    |   movel([0.686921, -1.277827, -2.632564, -0.801997, 1.570796, 2.257718],accel_mss,speed_ms,0,blend_radius_m)
    |   speed_ms = 0.040
    |   movel([0.686153, -1.291546, -2.624638, -0.796205, 1.570796, 2.256949],accel_mss,speed_ms,0,blend_radius_m)
    |   speed_ms = 0.005
    |   movel([0.686153, -1.300886, -2.628985, -0.782518, 1.570796, 2.256949],accel_mss,speed_ms,0,blend_radius_m)
    |   speed_ms = 0.025
    |   movel([0.686563, -1.298464, -2.630421, -0.783504, 1.570796, 2.257359],accel_mss,speed_ms,0,blend_radius_m)
    |   movel([0.686602, -1.296181, -2.631767, -0.784440, 1.570796, 2.257399],accel_mss,speed_ms,0,blend_radius_m)
    |   movel([0.686283, -1.294070, -2.633007, -0.785312, 1.570796, 2.257079],accel_mss,speed_ms,0,blend_radius_m)
    |   movel([0.685611, -1.292156, -2.634126, -0.786108, 1.570796, 2.256407],accel_mss,speed_ms,0,blend_radius_m)
    |   movel([0.684603, -1.290473, -2.635106, -0.786811, 1.570796, 2.255399],accel_mss,speed_ms,0,blend_radius_m)
    |   movel([0.683264, -1.289050, -2.635931, -0.787408, 1.570796, 2.254061],accel_mss,speed_ms,0,blend_radius_m)
    |   movel([0.681611, -1.287921, -2.636584, -0.787884, 1.570796, 2.252407],accel_mss,speed_ms,0,blend_radius_m)
    |   movel([0.679652, -1.287111, -2.637052, -0.788226, 1.570796, 2.250448],accel_mss,speed_ms,0,blend_radius_m)
    |   movel([0.677407, -1.286654, -2.637315, -0.788420, 1.570796, 2.248203],accel_mss,speed_ms,0,blend_radius_m)
    |   movel([0.674916, -1.286573, -2.637362, -0.788454, 1.570796, 2.245712],accel_mss,speed_ms,0,blend_radius_m)
    |   movel([0.672268, -1.286884, -2.637182, -0.788322, 1.570796, 2.243064],accel_mss,speed_ms,0,blend_radius_m)
    |   movel([0.669552, -1.287613, -2.636762, -0.788014, 1.570796, 2.240348],accel_mss,speed_ms,0,blend_radius_m)
    |   movel([0.666852, -1.288777, -2.636089, -0.787523, 1.570796, 2.237648],accel_mss,speed_ms,0,blend_radius_m)
    |   movel([0.665538, -1.289527, -2.635654, -0.787208, 1.570796, 2.236335],accel_mss,speed_ms,0,blend_radius_m)
    |   movel([0.664263, -1.290390, -2.635154, -0.786846, 1.570796, 2.235059],accel_mss,speed_ms,0,blend_radius_m)
    |   movel([0.663035, -1.291369, -2.634584, -0.786436, 1.570796, 2.233831],accel_mss,speed_ms,0,blend_radius_m)
    |   movel([0.661866, -1.292469, -2.633943, -0.785977, 1.570796, 2.232663],accel_mss,speed_ms,0,blend_radius_m)
    |   movel([0.660768, -1.293687, -2.633231, -0.785471, 1.570796, 2.231564],accel_mss,speed_ms,0,blend_radius_m)
    |   movel([0.659756, -1.295024, -2.632448, -0.784917, 1.570796, 2.230552],accel_mss,speed_ms,0,blend_radius_m)
    |   speed_ms = 0.005
    |   movel([0.659756, -1.285649, -2.628074, -0.798666, 1.570796, 2.230552],accel_mss,speed_ms,0,blend_radius_m)
    |   speed_ms = 0.040
    |   movel([0.667434, -1.296086, -2.621962, -0.794341, 1.570796, 2.238230],accel_mss,speed_ms,0,blend_radius_m)
    |   speed_ms = 0.005
    |   movel([0.667434, -1.305400, -2.626288, -0.780701, 1.570796, 2.238230],accel_mss,speed_ms,0,blend_radius_m)
    |   speed_ms = 0.025
    |   movel([0.669418, -1.304874, -2.626604, -0.780911, 1.570796, 2.240215],accel_mss,speed_ms,0,blend_radius_m)
    |   movel([0.671310, -1.304654, -2.626736, -0.781000, 1.570796, 2.242106],accel_mss,speed_ms,0,blend_radius_m)
    |   movel([0.673092, -1.304715, -2.626699, -0.780975, 1.570796, 2.243888],accel_mss,speed_ms,0,blend_radius_m)
    |   movel([0.674741, -1.305035, -2.626507, -0.780847, 1.570796, 2.245537],accel_mss,speed_ms,0,blend_radius_m)
    |   movel([0.676240, -1.305588, -2.626175, -0.780626, 1.570796, 2.247036],accel_mss,speed_ms,0,blend_radius_m)
    |   movel([0.677570, -1.306343, -2.625722, -0.780325, 1.570796, 2.248366],accel_mss,speed_ms,0,blend_radius_m)
    |   movel([0.678716, -1.307277, -2.625159, -0.779953, 1.570796, 2.249512],accel_mss,speed_ms,0,blend_radius_m)
    |   movel([0.679657, -1.308360, -2.624505, -0.779524, 1.570796, 2.250453],accel_mss,speed_ms,0,blend_radius_m)
    |   movel([0.680469, -1.309890, -2.623579, -0.778920, 1.570796, 2.251265],accel_mss,speed_ms,0,blend_radius_m)
    |   movel([0.680812, -1.311531, -2.622583, -0.778276, 1.570796, 2.251609],accel_mss,speed_ms,0,blend_radius_m)
    |   movel([0.680741, -1.313269, -2.621523, -0.777597, 1.570796, 2.251537],accel_mss,speed_ms,0,blend_radius_m)
    |   movel([0.680298, -1.315090, -2.620408, -0.776890, 1.570796, 2.251095],accel_mss,speed_ms,0,blend_radius_m)
    |   movel([0.679538, -1.316977, -2.619249, -0.776163, 1.570796, 2.250334],accel_mss,speed_ms,0,blend_radius_m)
    |   movel([0.678505, -1.318918, -2.618051, -0.775419, 1.570796, 2.249301],accel_mss,speed_ms,0,blend_radius_m)
    |   movel([0.677248, -1.320898, -2.616825, -0.774666, 1.570796, 2.248044],accel_mss,speed_ms,0,blend_radius_m)
    |   movel([0.675817, -1.322904, -2.615576, -0.773908, 1.570796, 2.246614],accel_mss,speed_ms,0,blend_radius_m)
    |   speed_ms = 0.005
    |   movel([0.675817, -1.313698, -2.611330, -0.787361, 1.570796, 2.246614],accel_mss,speed_ms,0,blend_radius_m)
    |   speed_ms = 0.040
    |   movel([0.665940, -1.309142, -2.614119, -0.789128, 1.570796, 2.236737],accel_mss,speed_ms,0,blend_radius_m)
    |   speed_ms = 0.005
    |   movel([0.665940, -1.318376, -2.618386, -0.775626, 1.570796, 2.236737],accel_mss,speed_ms,0,blend_radius_m)
    |   speed_ms = 0.025
    |   movel([0.667189, -1.319166, -2.617898, -0.775325, 1.570796, 2.237985],accel_mss,speed_ms,0,blend_radius_m)
    |   movel([0.668210, -1.320110, -2.617314, -0.774965, 1.570796, 2.239007],accel_mss,speed_ms,0,blend_radius_m)
    |   movel([0.669011, -1.321200, -2.616637, -0.774552, 1.570796, 2.239807],accel_mss,speed_ms,0,blend_radius_m)
    |   movel([0.669605, -1.322415, -2.615881, -0.774093, 1.570796, 2.240401],accel_mss,speed_ms,0,blend_radius_m)
    |   movel([0.670000, -1.323744, -2.615052, -0.773593, 1.570796, 2.240796],accel_mss,speed_ms,0,blend_radius_m)
    |   movel([0.670206, -1.325167, -2.614162, -0.773060, 1.570796, 2.241002],accel_mss,speed_ms,0,blend_radius_m)
    |   movel([0.670235, -1.326674, -2.613216, -0.772499, 1.570796, 2.241031],accel_mss,speed_ms,0,blend_radius_m)
    |   movel([0.670092, -1.328248, -2.612225, -0.771916, 1.570796, 2.240888],accel_mss,speed_ms,0,blend_radius_m)
    |   movel([0.669791, -1.329876, -2.611196, -0.771317, 1.570796, 2.240588],accel_mss,speed_ms,0,blend_radius_m)
    |   movel([0.669343, -1.331542, -2.610139, -0.770707, 1.570796, 2.240139],accel_mss,speed_ms,0,blend_radius_m)
    |   movel([0.668753, -1.333234, -2.609063, -0.770092, 1.570796, 2.239550],accel_mss,speed_ms,0,blend_radius_m)
    |   movel([0.668036, -1.334937, -2.607975, -0.769477, 1.570796, 2.238832],accel_mss,speed_ms,0,blend_radius_m)
    |   movel([0.667196, -1.336639, -2.606884, -0.768866, 1.570796, 2.237993],accel_mss,speed_ms,0,blend_radius_m)
    |   movel([0.665195, -1.339980, -2.604731, -0.767678, 1.570796, 2.235992],accel_mss,speed_ms,0,blend_radius_m)
    |   movel([0.664049, -1.341596, -2.603683, -0.767109, 1.570796, 2.234845],accel_mss,speed_ms,0,blend_radius_m)
    |   movel([0.664256, -1.341009, -2.604065, -0.767316, 1.570796, 2.235052],accel_mss,speed_ms,0,blend_radius_m)
    |   speed_ms = 0.005
    |   movel([0.664256, -1.331920, -2.599899, -0.780569, 1.570796, 2.235052],accel_mss,speed_ms,0,blend_radius_m)
    |   speed_ms = 0.040
    |   movel([0.669329, -1.341680, -2.593594, -0.777115, 1.570796, 2.240125],accel_mss,speed_ms,0,blend_radius_m)
    |   speed_ms = 0.005
    |   movel([0.669329, -1.350703, -2.597716, -0.763970, 1.570796, 2.240125],accel_mss,speed_ms,0,blend_radius_m)
    |   speed_ms = 0.025
    |   movel([0.667012, -1.352255, -2.596687, -0.763446, 1.570796, 2.237809],accel_mss,speed_ms,0,blend_radius_m)
    |   movel([0.664808, -1.353984, -2.595538, -0.762867, 1.570796, 2.235605],accel_mss,speed_ms,0,blend_radius_m)
    |   movel([0.662701, -1.355833, -2.594304, -0.762253, 1.570796, 2.233497],accel_mss,speed_ms,0,blend_radius_m)
    |   movel([0.660671, -1.357746, -2.593022, -0.761621, 1.570796, 2.231468],accel_mss,speed_ms,0,blend_radius_m)
    |   movel([0.658520, -1.359912, -2.591564, -0.760913, 1.570796, 2.229316],accel_mss,speed_ms,0,blend_radius_m)
    |   movel([0.657534, -1.361038, -2.590803, -0.760548, 1.570796, 2.228330],accel_mss,speed_ms,0,blend_radius_m)
    |   movel([0.656649, -1.362205, -2.590013, -0.760171, 1.570796, 2.227445],accel_mss,speed_ms,0,blend_radius_m)
    |   movel([0.655897, -1.363413, -2.589194, -0.759782, 1.570796, 2.226693],accel_mss,speed_ms,0,blend_radius_m)
    |   movel([0.655325, -1.364636, -2.588362, -0.759391, 1.570796, 2.226121],accel_mss,speed_ms,0,blend_radius_m)
    |   movel([0.654988, -1.365827, -2.587550, -0.759013, 1.570796, 2.225784],accel_mss,speed_ms,0,blend_radius_m)
    |   movel([0.654928, -1.366946, -2.586784, -0.758659, 1.570796, 2.225725],accel_mss,speed_ms,0,blend_radius_m)
    |   movel([0.655311, -1.368509, -2.585713, -0.758167, 1.570796, 2.226108],accel_mss,speed_ms,0,blend_radius_m)
    |   movel([0.655496, -1.369287, -2.585178, -0.757924, 1.570796, 2.226293],accel_mss,speed_ms,0,blend_radius_m)
    |   movel([0.655524, -1.370128, -2.584599, -0.757662, 1.570796, 2.226321],accel_mss,speed_ms,0,blend_radius_m)
    |   movel([0.655238, -1.371196, -2.583862, -0.757331, 1.570796, 2.226035],accel_mss,speed_ms,0,blend_radius_m)
    |   movel([0.654635, -1.372378, -2.583045, -0.756966, 1.570796, 2.225432],accel_mss,speed_ms,0,blend_radius_m)
    |   movel([0.653794, -1.373631, -2.582177, -0.756581, 1.570796, 2.224590],accel_mss,speed_ms,0,blend_radius_m)
    |   movel([0.652789, -1.374910, -2.581288, -0.756191, 1.570796, 2.223585],accel_mss,speed_ms,0,blend_radius_m)
    |   movel([0.650587, -1.377373, -2.579570, -0.755446, 1.570796, 2.221383],accel_mss,speed_ms,0,blend_radius_m)
    |   movel([0.644135, -1.383963, -2.574929, -0.753497, 1.570796, 2.214932],accel_mss,speed_ms,0,blend_radius_m)
    |   movel([0.639695, -1.388489, -2.571706, -0.752194, 1.570796, 2.210491],accel_mss,speed_ms,0,blend_radius_m)
    |   movel([0.638417, -1.389930, -2.570673, -0.751785, 1.570796, 2.209214],accel_mss,speed_ms,0,blend_radius_m)
    |   movel([0.637140, -1.391519, -2.569531, -0.751339, 1.570796, 2.207937],accel_mss,speed_ms,0,blend_radius_m)
    |   movel([0.634709, -1.395002, -2.567015, -0.750372, 1.570796, 2.205506],accel_mss,speed_ms,0,blend_radius_m)
    |   movel([0.633617, -1.396832, -2.565686, -0.749871, 1.570796, 2.204414],accel_mss,speed_ms,0,blend_radius_m)
    |   movel([0.632649, -1.398676, -2.564341, -0.749371, 1.570796, 2.203445],accel_mss,speed_ms,0,blend_radius_m)
    |   movel([0.631834, -1.400502, -2.563006, -0.748882, 1.570796, 2.202630],accel_mss,speed_ms,0,blend_radius_m)
    |   movel([0.631200, -1.402278, -2.561701, -0.748410, 1.570796, 2.201996],accel_mss,speed_ms,0,blend_radius_m)
    |   movel([0.630780, -1.403969, -2.560455, -0.747965, 1.570796, 2.201576],accel_mss,speed_ms,0,blend_radius_m)
    |   movel([0.630598, -1.405550, -2.559286, -0.747553, 1.570796, 2.201395],accel_mss,speed_ms,0,blend_radius_m)
    |   movel([0.630689, -1.406985, -2.558221, -0.747182, 1.570796, 2.201485],accel_mss,speed_ms,0,blend_radius_m)
    |   movel([0.631078, -1.408246, -2.557284, -0.746859, 1.570796, 2.201874],accel_mss,speed_ms,0,blend_radius_m)
    |   movel([0.631793, -1.409302, -2.556497, -0.746590, 1.570796, 2.202590],accel_mss,speed_ms,0,blend_radius_m)
    |   movel([0.632867, -1.410123, -2.555884, -0.746382, 1.570796, 2.203663],accel_mss,speed_ms,0,blend_radius_m)
    |   movel([0.634326, -1.410681, -2.555467, -0.746242, 1.570796, 2.205122],accel_mss,speed_ms,0,blend_radius_m)
    |   movel([0.636200, -1.410945, -2.555268, -0.746175, 1.570796, 2.206996],accel_mss,speed_ms,0,blend_radius_m)
    |   movel([0.637786, -1.410925, -2.555284, -0.746180, 1.570796, 2.208582],accel_mss,speed_ms,0,blend_radius_m)
    |   movel([0.639424, -1.410729, -2.555430, -0.746230, 1.570796, 2.210220],accel_mss,speed_ms,0,blend_radius_m)
    |   movel([0.641107, -1.410385, -2.555688, -0.746316, 1.570796, 2.211903],accel_mss,speed_ms,0,blend_radius_m)
    |   movel([0.642824, -1.409921, -2.556034, -0.746433, 1.570796, 2.213620],accel_mss,speed_ms,0,blend_radius_m)
    |   movel([0.646315, -1.408753, -2.556906, -0.746730, 1.570796, 2.217111],accel_mss,speed_ms,0,blend_radius_m)
    |   movel([0.649813, -1.407458, -2.557870, -0.747061, 1.570796, 2.220609],accel_mss,speed_ms,0,blend_radius_m)
    |   movel([0.653331, -1.406258, -2.558761, -0.747370, 1.570796, 2.224127],accel_mss,speed_ms,0,blend_radius_m)
    |   movel([0.655091, -1.405764, -2.559127, -0.747498, 1.570796, 2.225887],accel_mss,speed_ms,0,blend_radius_m)
    |   movel([0.656821, -1.405383, -2.559410, -0.747597, 1.570796, 2.227617],accel_mss,speed_ms,0,blend_radius_m)
    |   movel([0.658499, -1.405139, -2.559590, -0.747660, 1.570796, 2.229295],accel_mss,speed_ms,0,blend_radius_m)
    |   movel([0.660101, -1.405068, -2.559642, -0.747678, 1.570796, 2.230897],accel_mss,speed_ms,0,blend_radius_m)
    |   movel([0.661602, -1.405196, -2.559548, -0.747645, 1.570796, 2.232399],accel_mss,speed_ms,0,blend_radius_m)
    |   movel([0.662981, -1.405554, -2.559283, -0.747552, 1.570796, 2.233778],accel_mss,speed_ms,0,blend_radius_m)
    |   movel([0.665610, -1.406851, -2.558321, -0.747217, 1.570796, 2.236406],accel_mss,speed_ms,0,blend_radius_m)
    |   movel([0.666547, -1.407202, -2.558060, -0.747127, 1.570796, 2.237343],accel_mss,speed_ms,0,blend_radius_m)
    |   movel([0.667629, -1.407372, -2.557934, -0.747083, 1.570796, 2.238425],accel_mss,speed_ms,0,blend_radius_m)
    |   movel([0.668828, -1.407294, -2.557992, -0.747103, 1.570796, 2.239625],accel_mss,speed_ms,0,blend_radius_m)
    |   movel([0.670052, -1.406927, -2.558265, -0.747197, 1.570796, 2.240849],accel_mss,speed_ms,0,blend_radius_m)
    |   movel([0.670647, -1.406620, -2.558492, -0.747276, 1.570796, 2.241444],accel_mss,speed_ms,0,blend_radius_m)
    |   movel([0.671215, -1.406225, -2.558785, -0.747378, 1.570796, 2.242011],accel_mss,speed_ms,0,blend_radius_m)
    |   speed_ms = 0.005
    |   movel([0.671215, -1.397599, -2.554908, -0.759882, 1.570796, 2.242011],accel_mss,speed_ms,0,blend_radius_m)
    |   speed_ms = 0.040
    |   movel([0.680691, -1.388985, -2.561158, -0.762246, 1.570796, 2.251487],accel_mss,speed_ms,0,blend_radius_m)
    |   speed_ms = 0.005
    |   movel([0.680691, -1.397674, -2.565072, -0.749642, 1.570796, 2.251487],accel_mss,speed_ms,0,blend_radius_m)
    |   speed_ms = 0.025
    |   movel([0.680883, -1.398010, -2.564828, -0.749551, 1.570796, 2.251680],accel_mss,speed_ms,0,blend_radius_m)
    |   movel([0.680674, -1.398511, -2.564462, -0.749416, 1.570796, 2.251470],accel_mss,speed_ms,0,blend_radius_m)
    |   movel([0.680200, -1.399003, -2.564103, -0.749283, 1.570796, 2.250996],accel_mss,speed_ms,0,blend_radius_m)
    |   movel([0.679605, -1.399318, -2.563872, -0.749199, 1.570796, 2.250401],accel_mss,speed_ms,0,blend_radius_m)
    |   movel([0.679026, -1.399397, -2.563814, -0.749177, 1.570796, 2.249822],accel_mss,speed_ms,0,blend_radius_m)
    |   movel([0.678495, -1.399343, -2.563854, -0.749192, 1.570796, 2.249291],accel_mss,speed_ms,0,blend_radius_m)
    |   movel([0.677488, -1.399100, -2.564032, -0.749257, 1.570796, 2.248284],accel_mss,speed_ms,0,blend_radius_m)
    |   movel([0.676711, -1.399024, -2.564088, -0.749278, 1.570796, 2.247507],accel_mss,speed_ms,0,blend_radius_m)
    |   movel([0.675887, -1.399074, -2.564050, -0.749264, 1.570796, 2.246684],accel_mss,speed_ms,0,blend_radius_m)
    |   movel([0.674136, -1.399477, -2.563756, -0.749156, 1.570796, 2.244932],accel_mss,speed_ms,0,blend_radius_m)
    |   movel([0.672313, -1.400165, -2.563253, -0.748972, 1.570796, 2.243109],accel_mss,speed_ms,0,blend_radius_m)
    |   movel([0.670505, -1.400982, -2.562653, -0.748754, 1.570796, 2.241301],accel_mss,speed_ms,0,blend_radius_m)
    |   movel([0.670073, -1.401213, -2.562483, -0.748692, 1.570796, 2.240869],accel_mss,speed_ms,0,blend_radius_m)
    |   movel([0.669730, -1.401530, -2.562251, -0.748608, 1.570796, 2.240527],accel_mss,speed_ms,0,blend_radius_m)
    |   movel([0.669616, -1.401957, -2.561937, -0.748495, 1.570796, 2.240413],accel_mss,speed_ms,0,blend_radius_m)
    |   movel([0.669756, -1.402325, -2.561667, -0.748398, 1.570796, 2.240552],accel_mss,speed_ms,0,blend_radius_m)
    |   movel([0.670265, -1.402999, -2.561170, -0.748220, 1.570796, 2.241062],accel_mss,speed_ms,0,blend_radius_m)
    |   movel([0.670916, -1.403551, -2.560763, -0.748075, 1.570796, 2.241712],accel_mss,speed_ms,0,blend_radius_m)
    |   movel([0.671691, -1.403981, -2.560446, -0.747962, 1.570796, 2.242488],accel_mss,speed_ms,0,blend_radius_m)
    |   movel([0.672577, -1.404280, -2.560225, -0.747884, 1.570796, 2.243373],accel_mss,speed_ms,0,blend_radius_m)
    |   movel([0.673550, -1.404448, -2.560101, -0.747840, 1.570796, 2.244346],accel_mss,speed_ms,0,blend_radius_m)
    |   movel([0.674597, -1.404478, -2.560079, -0.747832, 1.570796, 2.245393],accel_mss,speed_ms,0,blend_radius_m)
    |   movel([0.675697, -1.404367, -2.560161, -0.747861, 1.570796, 2.246493],accel_mss,speed_ms,0,blend_radius_m)
    |   movel([0.676837, -1.404109, -2.560351, -0.747929, 1.570796, 2.247633],accel_mss,speed_ms,0,blend_radius_m)
    |   movel([0.676413, -1.404676, -2.559932, -0.747781, 1.570796, 2.247210],accel_mss,speed_ms,0,blend_radius_m)
    |   movel([0.676247, -1.405267, -2.559495, -0.747627, 1.570796, 2.247043],accel_mss,speed_ms,0,blend_radius_m)
    |   movel([0.676318, -1.405806, -2.559096, -0.747487, 1.570796, 2.247115],accel_mss,speed_ms,0,blend_radius_m)
    |   movel([0.676606, -1.406219, -2.558790, -0.747380, 1.570796, 2.247403],accel_mss,speed_ms,0,blend_radius_m)
    |   movel([0.677062, -1.406468, -2.558605, -0.747316, 1.570796, 2.247858],accel_mss,speed_ms,0,blend_radius_m)
    |   movel([0.677622, -1.406590, -2.558515, -0.747284, 1.570796, 2.248418],accel_mss,speed_ms,0,blend_radius_m)
    |   movel([0.678903, -1.406555, -2.558541, -0.747293, 1.570796, 2.249699],accel_mss,speed_ms,0,blend_radius_m)
    |   movel([0.680637, -1.406212, -2.558795, -0.747382, 1.570796, 2.251433],accel_mss,speed_ms,0,blend_radius_m)
    |   movel([0.682402, -1.405611, -2.559240, -0.747537, 1.570796, 2.253199],accel_mss,speed_ms,0,blend_radius_m)
    |   movel([0.684148, -1.404776, -2.559859, -0.747755, 1.570796, 2.254944],accel_mss,speed_ms,0,blend_radius_m)
    |   movel([0.685822, -1.403724, -2.560635, -0.748029, 1.570796, 2.256618],accel_mss,speed_ms,0,blend_radius_m)
    |   movel([0.686346, -1.403307, -2.560943, -0.748139, 1.570796, 2.257143],accel_mss,speed_ms,0,blend_radius_m)
    |   movel([0.686712, -1.402817, -2.561304, -0.748268, 1.570796, 2.257508],accel_mss,speed_ms,0,blend_radius_m)
    |   movel([0.686787, -1.402398, -2.561612, -0.748378, 1.570796, 2.257584],accel_mss,speed_ms,0,blend_radius_m)
    |   movel([0.686704, -1.402025, -2.561887, -0.748477, 1.570796, 2.257500],accel_mss,speed_ms,0,blend_radius_m)
    |   movel([0.686178, -1.400920, -2.562699, -0.748770, 1.570796, 2.256975],accel_mss,speed_ms,0,blend_radius_m)
    |   movel([0.684967, -1.399025, -2.564086, -0.749277, 1.570796, 2.255763],accel_mss,speed_ms,0,blend_radius_m)
    |   movel([0.684628, -1.397802, -2.564979, -0.749608, 1.570796, 2.255424],accel_mss,speed_ms,0,blend_radius_m)
    |   movel([0.686712, -1.396981, -2.565578, -0.749831, 1.570796, 2.257509],accel_mss,speed_ms,0,blend_radius_m)
    |   movel([0.687737, -1.396754, -2.565743, -0.749893, 1.570796, 2.258533],accel_mss,speed_ms,0,blend_radius_m)
    |   movel([0.688707, -1.396701, -2.565781, -0.749907, 1.570796, 2.259503],accel_mss,speed_ms,0,blend_radius_m)
    |   movel([0.689312, -1.396793, -2.565714, -0.749882, 1.570796, 2.260109],accel_mss,speed_ms,0,blend_radius_m)
    |   movel([0.689888, -1.396995, -2.565567, -0.749827, 1.570796, 2.260685],accel_mss,speed_ms,0,blend_radius_m)
    |   movel([0.690779, -1.397631, -2.565104, -0.749654, 1.570796, 2.261575],accel_mss,speed_ms,0,blend_radius_m)
    |   movel([0.691061, -1.398318, -2.564603, -0.749468, 1.570796, 2.261857],accel_mss,speed_ms,0,blend_radius_m)
    |   movel([0.691028, -1.398733, -2.564300, -0.749356, 1.570796, 2.261825],accel_mss,speed_ms,0,blend_radius_m)
    |   movel([0.690852, -1.399170, -2.563980, -0.749239, 1.570796, 2.261648],accel_mss,speed_ms,0,blend_radius_m)
    |   movel([0.690426, -1.399699, -2.563593, -0.749096, 1.570796, 2.261223],accel_mss,speed_ms,0,blend_radius_m)
    |   movel([0.689862, -1.400133, -2.563276, -0.748980, 1.570796, 2.260658],accel_mss,speed_ms,0,blend_radius_m)
    |   movel([0.688558, -1.400756, -2.562819, -0.748814, 1.570796, 2.259355],accel_mss,speed_ms,0,blend_radius_m)
    |   speed_ms = 0.005
    |   movel([0.688558, -1.392089, -2.558918, -0.761382, 1.570796, 2.259355],accel_mss,speed_ms,0,blend_radius_m)
    |   speed_ms = 0.040
    |   movel([0.716496, -1.351915, -2.586842, -0.773633, 1.570796, 2.287292],accel_mss,speed_ms,0,blend_radius_m)
    |   speed_ms = 0.005
    |   movel([0.716496, -1.360868, -2.590918, -0.760603, 1.570796, 2.287292],accel_mss,speed_ms,0,blend_radius_m)
    |   speed_ms = 0.025
    |   movel([0.717258, -1.360764, -2.590989, -0.760636, 1.570796, 2.288054],accel_mss,speed_ms,0,blend_radius_m)
    |   movel([0.717956, -1.360800, -2.590965, -0.760625, 1.570796, 2.288752],accel_mss,speed_ms,0,blend_radius_m)
    |   movel([0.718581, -1.360962, -2.590855, -0.760572, 1.570796, 2.289378],accel_mss,speed_ms,0,blend_radius_m)
    |   movel([0.719585, -1.361618, -2.590411, -0.760360, 1.570796, 2.290381],accel_mss,speed_ms,0,blend_radius_m)
    |   movel([0.719948, -1.362084, -2.590096, -0.760210, 1.570796, 2.290744],accel_mss,speed_ms,0,blend_radius_m)
    |   movel([0.720357, -1.363222, -2.589323, -0.759844, 1.570796, 2.291153],accel_mss,speed_ms,0,blend_radius_m)
    |   movel([0.720360, -1.364536, -2.588430, -0.759423, 1.570796, 2.291156],accel_mss,speed_ms,0,blend_radius_m)
    |   movel([0.720047, -1.365943, -2.587470, -0.758976, 1.570796, 2.290843],accel_mss,speed_ms,0,blend_radius_m)
    |   movel([0.719489, -1.367396, -2.586476, -0.758517, 1.570796, 2.290286],accel_mss,speed_ms,0,blend_radius_m)
    |   movel([0.718758, -1.368847, -2.585480, -0.758061, 1.570796, 2.289554],accel_mss,speed_ms,0,blend_radius_m)
    |   movel([0.717424, -1.371005, -2.583994, -0.757390, 1.570796, 2.288221],accel_mss,speed_ms,0,blend_radius_m)
    |   movel([0.715860, -1.373097, -2.582547, -0.756745, 1.570796, 2.286657],accel_mss,speed_ms,0,blend_radius_m)
    |   movel([0.714092, -1.375092, -2.581162, -0.756136, 1.570796, 2.284888],accel_mss,speed_ms,0,blend_radius_m)
    |   movel([0.710270, -1.378698, -2.578642, -0.755049, 1.570796, 2.281067],accel_mss,speed_ms,0,blend_radius_m)
    |   movel([0.709523, -1.379622, -2.577993, -0.754774, 1.570796, 2.280320],accel_mss,speed_ms,0,blend_radius_m)
    |   movel([0.709071, -1.380588, -2.577314, -0.754487, 1.570796, 2.279868],accel_mss,speed_ms,0,blend_radius_m)
    |   movel([0.709002, -1.381412, -2.576733, -0.754244, 1.570796, 2.279798],accel_mss,speed_ms,0,blend_radius_m)
    |   movel([0.709144, -1.382165, -2.576202, -0.754022, 1.570796, 2.279941],accel_mss,speed_ms,0,blend_radius_m)
    |   movel([0.709330, -1.382908, -2.575677, -0.753805, 1.570796, 2.280126],accel_mss,speed_ms,0,blend_radius_m)
    |   movel([0.709385, -1.383698, -2.575117, -0.753574, 1.570796, 2.280182],accel_mss,speed_ms,0,blend_radius_m)
    |   movel([0.709218, -1.384465, -2.574573, -0.753351, 1.570796, 2.280015],accel_mss,speed_ms,0,blend_radius_m)
    |   movel([0.708871, -1.385254, -2.574013, -0.753122, 1.570796, 2.279667],accel_mss,speed_ms,0,blend_radius_m)
    |   movel([0.707876, -1.386827, -2.572893, -0.752669, 1.570796, 2.278672],accel_mss,speed_ms,0,blend_radius_m)
    |   movel([0.706251, -1.389023, -2.571323, -0.752042, 1.570796, 2.277047],accel_mss,speed_ms,0,blend_radius_m)
    |   movel([0.704515, -1.391169, -2.569783, -0.751437, 1.570796, 2.275312],accel_mss,speed_ms,0,blend_radius_m)
    |   movel([0.702673, -1.393253, -2.568281, -0.750855, 1.570796, 2.273470],accel_mss,speed_ms,0,blend_radius_m)
    |   movel([0.700734, -1.395274, -2.566818, -0.750297, 1.570796, 2.271531],accel_mss,speed_ms,0,blend_radius_m)
    |   movel([0.698706, -1.397219, -2.565404, -0.749766, 1.570796, 2.269502],accel_mss,speed_ms,0,blend_radius_m)
    |   movel([0.696598, -1.399086, -2.564042, -0.749261, 1.570796, 2.267395],accel_mss,speed_ms,0,blend_radius_m)
    |   movel([0.694414, -1.400865, -2.562739, -0.748785, 1.570796, 2.265210],accel_mss,speed_ms,0,blend_radius_m)
    |   movel([0.692163, -1.402553, -2.561498, -0.748337, 1.570796, 2.262959],accel_mss,speed_ms,0,blend_radius_m)
    |   movel([0.690695, -1.403546, -2.560767, -0.748076, 1.570796, 2.261491],accel_mss,speed_ms,0,blend_radius_m)
    |   movel([0.689166, -1.404397, -2.560139, -0.747853, 1.570796, 2.259962],accel_mss,speed_ms,0,blend_radius_m)
    |   movel([0.687647, -1.404971, -2.559714, -0.747704, 1.570796, 2.258444],accel_mss,speed_ms,0,blend_radius_m)
    |   movel([0.686916, -1.405108, -2.559613, -0.747668, 1.570796, 2.257712],accel_mss,speed_ms,0,blend_radius_m)
    |   movel([0.686211, -1.405127, -2.559599, -0.747663, 1.570796, 2.257008],accel_mss,speed_ms,0,blend_radius_m)
    |   speed_ms = 0.005
    |   movel([0.686211, -1.396492, -2.555717, -0.760179, 1.570796, 2.257008],accel_mss,speed_ms,0,blend_radius_m)
    |   speed_ms = 0.040
    |   movel([0.681592, -1.398702, -2.554100, -0.759587, 1.570796, 2.252389],accel_mss,speed_ms,0,blend_radius_m)
    |   speed_ms = 0.005
    |   movel([0.681592, -1.407320, -2.557973, -0.747096, 1.570796, 2.252389],accel_mss,speed_ms,0,blend_radius_m)
    |   speed_ms = 0.025
    |   movel([0.681484, -1.407835, -2.557590, -0.746964, 1.570796, 2.252280],accel_mss,speed_ms,0,blend_radius_m)
    |   movel([0.681136, -1.408357, -2.557201, -0.746831, 1.570796, 2.251933],accel_mss,speed_ms,0,blend_radius_m)
    |   movel([0.680630, -1.408828, -2.556850, -0.746711, 1.570796, 2.251426],accel_mss,speed_ms,0,blend_radius_m)
    |   movel([0.680041, -1.409185, -2.556584, -0.746620, 1.570796, 2.250837],accel_mss,speed_ms,0,blend_radius_m)
    |   movel([0.679332, -1.409393, -2.556429, -0.746567, 1.570796, 2.250129],accel_mss,speed_ms,0,blend_radius_m)
    |   movel([0.678677, -1.409430, -2.556402, -0.746558, 1.570796, 2.249473],accel_mss,speed_ms,0,blend_radius_m)
    |   movel([0.678045, -1.409441, -2.556393, -0.746555, 1.570796, 2.248841],accel_mss,speed_ms,0,blend_radius_m)
    |   movel([0.677412, -1.409578, -2.556291, -0.746520, 1.570796, 2.248209],accel_mss,speed_ms,0,blend_radius_m)
    |   movel([0.676574, -1.410138, -2.555872, -0.746378, 1.570796, 2.247371],accel_mss,speed_ms,0,blend_radius_m)
    |   movel([0.676161, -1.410463, -2.555630, -0.746297, 1.570796, 2.246957],accel_mss,speed_ms,0,blend_radius_m)
    |   movel([0.675669, -1.410734, -2.555427, -0.746228, 1.570796, 2.246466],accel_mss,speed_ms,0,blend_radius_m)
    |   movel([0.674291, -1.411191, -2.555085, -0.746113, 1.570796, 2.245087],accel_mss,speed_ms,0,blend_radius_m)
    |   movel([0.672989, -1.411429, -2.554907, -0.746054, 1.570796, 2.243785],accel_mss,speed_ms,0,blend_radius_m)
    |   movel([0.671745, -1.411471, -2.554875, -0.746043, 1.570796, 2.242541],accel_mss,speed_ms,0,blend_radius_m)
    |   movel([0.670537, -1.411352, -2.554964, -0.746073, 1.570796, 2.241333],accel_mss,speed_ms,0,blend_radius_m)
    |   movel([0.671198, -1.411343, -2.554971, -0.746075, 1.570796, 2.241994],accel_mss,speed_ms,0,blend_radius_m)
    |   movel([0.671802, -1.411437, -2.554900, -0.746052, 1.570796, 2.242598],accel_mss,speed_ms,0,blend_radius_m)
    |   movel([0.672251, -1.411733, -2.554679, -0.745978, 1.570796, 2.243048],accel_mss,speed_ms,0,blend_radius_m)
    |   movel([0.672389, -1.412243, -2.554296, -0.745850, 1.570796, 2.243185],accel_mss,speed_ms,0,blend_radius_m)
    |   movel([0.672121, -1.412850, -2.553840, -0.745699, 1.570796, 2.242917],accel_mss,speed_ms,0,blend_radius_m)
    |   movel([0.671586, -1.413396, -2.553429, -0.745563, 1.570796, 2.242382],accel_mss,speed_ms,0,blend_radius_m)
    |   movel([0.670928, -1.413792, -2.553132, -0.745466, 1.570796, 2.241724],accel_mss,speed_ms,0,blend_radius_m)
    |   movel([0.669125, -1.414418, -2.552660, -0.745311, 1.570796, 2.239921],accel_mss,speed_ms,0,blend_radius_m)
    |   movel([0.668030, -1.414636, -2.552495, -0.745257, 1.570796, 2.238827],accel_mss,speed_ms,0,blend_radius_m)
    |   movel([0.666973, -1.414730, -2.552425, -0.745234, 1.570796, 2.237769],accel_mss,speed_ms,0,blend_radius_m)
    |   movel([0.665965, -1.414695, -2.552451, -0.745243, 1.570796, 2.236761],accel_mss,speed_ms,0,blend_radius_m)
    |   movel([0.667027, -1.414906, -2.552292, -0.745191, 1.570796, 2.237823],accel_mss,speed_ms,0,blend_radius_m)
    |   movel([0.668207, -1.414974, -2.552241, -0.745174, 1.570796, 2.239003],accel_mss,speed_ms,0,blend_radius_m)
    |   movel([0.669347, -1.415067, -2.552171, -0.745152, 1.570796, 2.240143],accel_mss,speed_ms,0,blend_radius_m)
    |   movel([0.670300, -1.415343, -2.551962, -0.745084, 1.570796, 2.241096],accel_mss,speed_ms,0,blend_radius_m)
    |   movel([0.670495, -1.415563, -2.551796, -0.745030, 1.570796, 2.241292],accel_mss,speed_ms,0,blend_radius_m)
    |   movel([0.670387, -1.415809, -2.551610, -0.744970, 1.570796, 2.241183],accel_mss,speed_ms,0,blend_radius_m)
    |   movel([0.669406, -1.416589, -2.551020, -0.744780, 1.570796, 2.240202],accel_mss,speed_ms,0,blend_radius_m)
    |   movel([0.668616, -1.417053, -2.550668, -0.744667, 1.570796, 2.239412],accel_mss,speed_ms,0,blend_radius_m)
    |   movel([0.667800, -1.417424, -2.550387, -0.744578, 1.570796, 2.238597],accel_mss,speed_ms,0,blend_radius_m)
    |   movel([0.666980, -1.417690, -2.550186, -0.744513, 1.570796, 2.237776],accel_mss,speed_ms,0,blend_radius_m)
    |   movel([0.667350, -1.417655, -2.550212, -0.744522, 1.570796, 2.238146],accel_mss,speed_ms,0,blend_radius_m)
    |   movel([0.667708, -1.417732, -2.550154, -0.744503, 1.570796, 2.238504],accel_mss,speed_ms,0,blend_radius_m)
    |   movel([0.668364, -1.418161, -2.549828, -0.744400, 1.570796, 2.239161],accel_mss,speed_ms,0,blend_radius_m)
    |   movel([0.668893, -1.418849, -2.549306, -0.744235, 1.570796, 2.239689],accel_mss,speed_ms,0,blend_radius_m)
    |   movel([0.669242, -1.419671, -2.548679, -0.744038, 1.570796, 2.240039],accel_mss,speed_ms,0,blend_radius_m)
    |   movel([0.669361, -1.420504, -2.548044, -0.743840, 1.570796, 2.240158],accel_mss,speed_ms,0,blend_radius_m)
    |   movel([0.669200, -1.421221, -2.547497, -0.743671, 1.570796, 2.239996],accel_mss,speed_ms,0,blend_radius_m)
    |   movel([0.668998, -1.421497, -2.547287, -0.743606, 1.570796, 2.239794],accel_mss,speed_ms,0,blend_radius_m)
    |   movel([0.668707, -1.421695, -2.547135, -0.743559, 1.570796, 2.239503],accel_mss,speed_ms,0,blend_radius_m)
    |   movel([0.668320, -1.421806, -2.547050, -0.743533, 1.570796, 2.239116],accel_mss,speed_ms,0,blend_radius_m)
    |   movel([0.667830, -1.421808, -2.547049, -0.743532, 1.570796, 2.238627],accel_mss,speed_ms,0,blend_radius_m)
    |   movel([0.667360, -1.421656, -2.547165, -0.743568, 1.570796, 2.238156],accel_mss,speed_ms,0,blend_radius_m)
    |   movel([0.665959, -1.420331, -2.548177, -0.743881, 1.570796, 2.236755],accel_mss,speed_ms,0,blend_radius_m)
    |   movel([0.665389, -1.419864, -2.548533, -0.743992, 1.570796, 2.236185],accel_mss,speed_ms,0,blend_radius_m)
    |   movel([0.664698, -1.419529, -2.548788, -0.744072, 1.570796, 2.235494],accel_mss,speed_ms,0,blend_radius_m)
    |   movel([0.663302, -1.419335, -2.548935, -0.744118, 1.570796, 2.234098],accel_mss,speed_ms,0,blend_radius_m)
    |   movel([0.661839, -1.419247, -2.549002, -0.744139, 1.570796, 2.232635],accel_mss,speed_ms,0,blend_radius_m)
    |   movel([0.661170, -1.419073, -2.549135, -0.744181, 1.570796, 2.231967],accel_mss,speed_ms,0,blend_radius_m)
    |   movel([0.660624, -1.418750, -2.549380, -0.744258, 1.570796, 2.231421],accel_mss,speed_ms,0,blend_radius_m)
    |   movel([0.660291, -1.418274, -2.549742, -0.744373, 1.570796, 2.231087],accel_mss,speed_ms,0,blend_radius_m)
    |   movel([0.660256, -1.417644, -2.550221, -0.744525, 1.570796, 2.231053],accel_mss,speed_ms,0,blend_radius_m)
    |   movel([0.661222, -1.417167, -2.550582, -0.744640, 1.570796, 2.232018],accel_mss,speed_ms,0,blend_radius_m)
    |   movel([0.662202, -1.416795, -2.550864, -0.744730, 1.570796, 2.232998],accel_mss,speed_ms,0,blend_radius_m)
    |   speed_ms = 0.005
    |   movel([0.662202, -1.408248, -2.547033, -0.757108, 1.570796, 2.232998],accel_mss,speed_ms,0,blend_radius_m)
    |   speed_ms = 0.040
    |   movel([0.664688, -1.417771, -2.539849, -0.754769, 1.570796, 2.235485],accel_mss,speed_ms,0,blend_radius_m)
    |   speed_ms = 0.005
    |   movel([0.664688, -1.426245, -2.543640, -0.742504, 1.570796, 2.235485],accel_mss,speed_ms,0,blend_radius_m)
    |   speed_ms = 0.025
    |   movel([0.665369, -1.425897, -2.543909, -0.742584, 1.570796, 2.236165],accel_mss,speed_ms,0,blend_radius_m)
    |   movel([0.666044, -1.425831, -2.543959, -0.742599, 1.570796, 2.236840],accel_mss,speed_ms,0,blend_radius_m)
    |   movel([0.666624, -1.426009, -2.543822, -0.742558, 1.570796, 2.237420],accel_mss,speed_ms,0,blend_radius_m)
    |   movel([0.667013, -1.426392, -2.543527, -0.742470, 1.570796, 2.237809],accel_mss,speed_ms,0,blend_radius_m)
    |   movel([0.667181, -1.426909, -2.543127, -0.742352, 1.570796, 2.237977],accel_mss,speed_ms,0,blend_radius_m)
    |   movel([0.667197, -1.427498, -2.542672, -0.742219, 1.570796, 2.237994],accel_mss,speed_ms,0,blend_radius_m)
    |   movel([0.666976, -1.428767, -2.541689, -0.741933, 1.570796, 2.237773],accel_mss,speed_ms,0,blend_radius_m)
    |   movel([0.667693, -1.428202, -2.542127, -0.742060, 1.570796, 2.238489],accel_mss,speed_ms,0,blend_radius_m)
    |   movel([0.668275, -1.427528, -2.542649, -0.742212, 1.570796, 2.239072],accel_mss,speed_ms,0,blend_radius_m)
    |   movel([0.668676, -1.426804, -2.543208, -0.742376, 1.570796, 2.239473],accel_mss,speed_ms,0,blend_radius_m)
    |   movel([0.668860, -1.426086, -2.543763, -0.742540, 1.570796, 2.239657],accel_mss,speed_ms,0,blend_radius_m)
    |   movel([0.669018, -1.426552, -2.543403, -0.742434, 1.570796, 2.239814],accel_mss,speed_ms,0,blend_radius_m)
    |   movel([0.669052, -1.427067, -2.543005, -0.742317, 1.570796, 2.239849],accel_mss,speed_ms,0,blend_radius_m)
    |   movel([0.668825, -1.428197, -2.542131, -0.742061, 1.570796, 2.239621],accel_mss,speed_ms,0,blend_radius_m)
    |   movel([0.668329, -1.429399, -2.541199, -0.741791, 1.570796, 2.239126],accel_mss,speed_ms,0,blend_radius_m)
    |   movel([0.667701, -1.430598, -2.540267, -0.741524, 1.570796, 2.238498],accel_mss,speed_ms,0,blend_radius_m)
    |   movel([0.666855, -1.431859, -2.539285, -0.741245, 1.570796, 2.237652],accel_mss,speed_ms,0,blend_radius_m)
    |   movel([0.665898, -1.432984, -2.538406, -0.740999, 1.570796, 2.236695],accel_mss,speed_ms,0,blend_radius_m)
    |   movel([0.664935, -1.434075, -2.537552, -0.740762, 1.570796, 2.235731],accel_mss,speed_ms,0,blend_radius_m)
    |   movel([0.664067, -1.435237, -2.536641, -0.740511, 1.570796, 2.234863],accel_mss,speed_ms,0,blend_radius_m)
    |   movel([0.664043, -1.434226, -2.537434, -0.740729, 1.570796, 2.234840],accel_mss,speed_ms,0,blend_radius_m)
    |   movel([0.663758, -1.433339, -2.538128, -0.740922, 1.570796, 2.234554],accel_mss,speed_ms,0,blend_radius_m)
    |   movel([0.663211, -1.432622, -2.538689, -0.741078, 1.570796, 2.234007],accel_mss,speed_ms,0,blend_radius_m)
    |   movel([0.662396, -1.432118, -2.539083, -0.741188, 1.570796, 2.233192],accel_mss,speed_ms,0,blend_radius_m)
    |   speed_ms = 0.005
    |   movel([0.662396, -1.423689, -2.535316, -0.753383, 1.570796, 2.233192],accel_mss,speed_ms,0,blend_radius_m)
    |   speed_ms = 0.040
    |   movel([0.661287, -1.428317, -2.531736, -0.752336, 1.570796, 2.232084],accel_mss,speed_ms,0,blend_radius_m)
    |   speed_ms = 0.005
    |   movel([0.661287, -1.436710, -2.535482, -0.740196, 1.570796, 2.232084],accel_mss,speed_ms,0,blend_radius_m)
    |   speed_ms = 0.025
    |   movel([0.660627, -1.438429, -2.534126, -0.739833, 1.570796, 2.231423],accel_mss,speed_ms,0,blend_radius_m)
    |   movel([0.660227, -1.440114, -2.532793, -0.739482, 1.570796, 2.231023],accel_mss,speed_ms,0,blend_radius_m)
    |   movel([0.660219, -1.441654, -2.531571, -0.739164, 1.570796, 2.231015],accel_mss,speed_ms,0,blend_radius_m)
    |   movel([0.660404, -1.442336, -2.531028, -0.739025, 1.570796, 2.231200],accel_mss,speed_ms,0,blend_radius_m)
    |   movel([0.660736, -1.442944, -2.530544, -0.738901, 1.570796, 2.231533],accel_mss,speed_ms,0,blend_radius_m)
    |   movel([0.661424, -1.443605, -2.530016, -0.738767, 1.570796, 2.232220],accel_mss,speed_ms,0,blend_radius_m)
    |   movel([0.662303, -1.444056, -2.529656, -0.738676, 1.570796, 2.233099],accel_mss,speed_ms,0,blend_radius_m)
    |   movel([0.663331, -1.444348, -2.529423, -0.738618, 1.570796, 2.234127],accel_mss,speed_ms,0,blend_radius_m)
    |   movel([0.664463, -1.444529, -2.529278, -0.738581, 1.570796, 2.235259],accel_mss,speed_ms,0,blend_radius_m)
    |   movel([0.666867, -1.444756, -2.529097, -0.738536, 1.570796, 2.237663],accel_mss,speed_ms,0,blend_radius_m)
    |   movel([0.669163, -1.445132, -2.528797, -0.738461, 1.570796, 2.239959],accel_mss,speed_ms,0,blend_radius_m)
    |   movel([0.670320, -1.445571, -2.528445, -0.738373, 1.570796, 2.241116],accel_mss,speed_ms,0,blend_radius_m)
    |   movel([0.671306, -1.446202, -2.527939, -0.738248, 1.570796, 2.242103],accel_mss,speed_ms,0,blend_radius_m)
    |   movel([0.672112, -1.447001, -2.527298, -0.738090, 1.570796, 2.242908],accel_mss,speed_ms,0,blend_radius_m)
    |   movel([0.672723, -1.447947, -2.526537, -0.737905, 1.570796, 2.243519],accel_mss,speed_ms,0,blend_radius_m)
    |   movel([0.673133, -1.449017, -2.525675, -0.737697, 1.570796, 2.243929],accel_mss,speed_ms,0,blend_radius_m)
    |   movel([0.673330, -1.450191, -2.524728, -0.737471, 1.570796, 2.244127],accel_mss,speed_ms,0,blend_radius_m)
    |   movel([0.673304, -1.451443, -2.523714, -0.737231, 1.570796, 2.244100],accel_mss,speed_ms,0,blend_radius_m)
    |   movel([0.673047, -1.452753, -2.522652, -0.736984, 1.570796, 2.243843],accel_mss,speed_ms,0,blend_radius_m)
    |   speed_ms = 0.005
    |   movel([0.673047, -1.444485, -2.518973, -0.748931, 1.570796, 2.243843],accel_mss,speed_ms,0,blend_radius_m)
    |   speed_ms = 0.040
    |   movel([0.663920, -1.413806, -2.542857, -0.755727, 1.570796, 2.234716],accel_mss,speed_ms,0,blend_radius_m)
    |   speed_ms = 0.005
    |   movel([0.663920, -1.422310, -2.546665, -0.743415, 1.570796, 2.234716],accel_mss,speed_ms,0,blend_radius_m)
    |   speed_ms = 0.025
    |   movel([0.664232, -1.422921, -2.546196, -0.743272, 1.570796, 2.235028],accel_mss,speed_ms,0,blend_radius_m)
    |   movel([0.664331, -1.423633, -2.545650, -0.743106, 1.570796, 2.235127],accel_mss,speed_ms,0,blend_radius_m)
    |   movel([0.664224, -1.424041, -2.545337, -0.743011, 1.570796, 2.235020],accel_mss,speed_ms,0,blend_radius_m)
    |   movel([0.663991, -1.424450, -2.545022, -0.742916, 1.570796, 2.234787],accel_mss,speed_ms,0,blend_radius_m)
    |   movel([0.663653, -1.424811, -2.544745, -0.742833, 1.570796, 2.234450],accel_mss,speed_ms,0,blend_radius_m)
    |   movel([0.663230, -1.425069, -2.544547, -0.742774, 1.570796, 2.234026],accel_mss,speed_ms,0,blend_radius_m)
    |   movel([0.662403, -1.425335, -2.544341, -0.742712, 1.570796, 2.233199],accel_mss,speed_ms,0,blend_radius_m)
    |   movel([0.662023, -1.425608, -2.544131, -0.742650, 1.570796, 2.232820],accel_mss,speed_ms,0,blend_radius_m)
    |   movel([0.661744, -1.425968, -2.543853, -0.742567, 1.570796, 2.232541],accel_mss,speed_ms,0,blend_radius_m)
    |   movel([0.661445, -1.426772, -2.543234, -0.742384, 1.570796, 2.232241],accel_mss,speed_ms,0,blend_radius_m)
    |   movel([0.661342, -1.427671, -2.542538, -0.742180, 1.570796, 2.232138],accel_mss,speed_ms,0,blend_radius_m)
    |   movel([0.661395, -1.428517, -2.541883, -0.741989, 1.570796, 2.232191],accel_mss,speed_ms,0,blend_radius_m)
    |   movel([0.661599, -1.429298, -2.541277, -0.741814, 1.570796, 2.232395],accel_mss,speed_ms,0,blend_radius_m)
    |   movel([0.661952, -1.429992, -2.540738, -0.741659, 1.570796, 2.232748],accel_mss,speed_ms,0,blend_radius_m)
    |   movel([0.661095, -1.430599, -2.540266, -0.741524, 1.570796, 2.231892],accel_mss,speed_ms,0,blend_radius_m)
    |   movel([0.660340, -1.431290, -2.539728, -0.741371, 1.570796, 2.231136],accel_mss,speed_ms,0,blend_radius_m)
    |   movel([0.659675, -1.432049, -2.539137, -0.741204, 1.570796, 2.230471],accel_mss,speed_ms,0,blend_radius_m)
    |   movel([0.659092, -1.432858, -2.538505, -0.741027, 1.570796, 2.229889],accel_mss,speed_ms,0,blend_radius_m)
    |   movel([0.658145, -1.434563, -2.537170, -0.740656, 1.570796, 2.228941],accel_mss,speed_ms,0,blend_radius_m)
    |   movel([0.657439, -1.436280, -2.535821, -0.740288, 1.570796, 2.228235],accel_mss,speed_ms,0,blend_radius_m)
    |   movel([0.656789, -1.437938, -2.534515, -0.739937, 1.570796, 2.227585],accel_mss,speed_ms,0,blend_radius_m)
    |   movel([0.656351, -1.438748, -2.533874, -0.739766, 1.570796, 2.227147],accel_mss,speed_ms,0,blend_radius_m)
    |   movel([0.655772, -1.439524, -2.533261, -0.739604, 1.570796, 2.226568],accel_mss,speed_ms,0,blend_radius_m)
    |   movel([0.654998, -1.440214, -2.532714, -0.739461, 1.570796, 2.225794],accel_mss,speed_ms,0,blend_radius_m)
    |   movel([0.654099, -1.440724, -2.532309, -0.739356, 1.570796, 2.224896],accel_mss,speed_ms,0,blend_radius_m)
    |   movel([0.653206, -1.440962, -2.532120, -0.739306, 1.570796, 2.224002],accel_mss,speed_ms,0,blend_radius_m)
    |   movel([0.652455, -1.440836, -2.532220, -0.739332, 1.570796, 2.223251],accel_mss,speed_ms,0,blend_radius_m)
    |   movel([0.652404, -1.441597, -2.531616, -0.739176, 1.570796, 2.223200],accel_mss,speed_ms,0,blend_radius_m)
    |   movel([0.651952, -1.443186, -2.530350, -0.738852, 1.570796, 2.222748],accel_mss,speed_ms,0,blend_radius_m)
    |   movel([0.651563, -1.443989, -2.529710, -0.738690, 1.570796, 2.222359],accel_mss,speed_ms,0,blend_radius_m)
    |   movel([0.650501, -1.445544, -2.528467, -0.738379, 1.570796, 2.221298],accel_mss,speed_ms,0,blend_radius_m)
    |   movel([0.649842, -1.446269, -2.527885, -0.738235, 1.570796, 2.220639],accel_mss,speed_ms,0,blend_radius_m)
    |   movel([0.649105, -1.446945, -2.527343, -0.738101, 1.570796, 2.219901],accel_mss,speed_ms,0,blend_radius_m)
    |   speed_ms = 0.005
    |   movel([0.649105, -1.438632, -2.523639, -0.750118, 1.570796, 2.219901],accel_mss,speed_ms,0,blend_radius_m)
    |   speed_ms = 0.040
    |   movel([0.645760, -1.437267, -2.524720, -0.750402, 1.570796, 2.216557],accel_mss,speed_ms,0,blend_radius_m)
    |   speed_ms = 0.005
    |   movel([0.645760, -1.445590, -2.528429, -0.738369, 1.570796, 2.216557],accel_mss,speed_ms,0,blend_radius_m)
    |   speed_ms = 0.025
    |   movel([0.643810, -1.453903, -2.521717, -0.736769, 1.570796, 2.214606],accel_mss,speed_ms,0,blend_radius_m)
    |   movel([0.643464, -1.454925, -2.520884, -0.736580, 1.570796, 2.214260],accel_mss,speed_ms,0,blend_radius_m)
    |   movel([0.643151, -1.455399, -2.520497, -0.736492, 1.570796, 2.213947],accel_mss,speed_ms,0,blend_radius_m)
    |   movel([0.642699, -1.455792, -2.520177, -0.736420, 1.570796, 2.213495],accel_mss,speed_ms,0,blend_radius_m)
    |   movel([0.641540, -1.456395, -2.519684, -0.736310, 1.570796, 2.212337],accel_mss,speed_ms,0,blend_radius_m)
    |   movel([0.641136, -1.456885, -2.519283, -0.736221, 1.570796, 2.211932],accel_mss,speed_ms,0,blend_radius_m)
    |   movel([0.640933, -1.457428, -2.518838, -0.736122, 1.570796, 2.211729],accel_mss,speed_ms,0,blend_radius_m)
    |   movel([0.640880, -1.458294, -2.518128, -0.735967, 1.570796, 2.211677],accel_mss,speed_ms,0,blend_radius_m)
    |   movel([0.641074, -1.459107, -2.517461, -0.735821, 1.570796, 2.211871],accel_mss,speed_ms,0,blend_radius_m)
    |   movel([0.641650, -1.460607, -2.516226, -0.735556, 1.570796, 2.212446],accel_mss,speed_ms,0,blend_radius_m)
    |   movel([0.641815, -1.461695, -2.515328, -0.735366, 1.570796, 2.212611],accel_mss,speed_ms,0,blend_radius_m)
    |   movel([0.641805, -1.463314, -2.513989, -0.735086, 1.570796, 2.212602],accel_mss,speed_ms,0,blend_radius_m)
    |   movel([0.641650, -1.464070, -2.513362, -0.734957, 1.570796, 2.212446],accel_mss,speed_ms,0,blend_radius_m)
    |   movel([0.641354, -1.464657, -2.512875, -0.734857, 1.570796, 2.212150],accel_mss,speed_ms,0,blend_radius_m)
    |   movel([0.641142, -1.464854, -2.512711, -0.734824, 1.570796, 2.211938],accel_mss,speed_ms,0,blend_radius_m)
    |   movel([0.640882, -1.464971, -2.512614, -0.734804, 1.570796, 2.211678],accel_mss,speed_ms,0,blend_radius_m)
    |   movel([0.640198, -1.464916, -2.512660, -0.734813, 1.570796, 2.210994],accel_mss,speed_ms,0,blend_radius_m)
    |   movel([0.639955, -1.465557, -2.512127, -0.734705, 1.570796, 2.210751],accel_mss,speed_ms,0,blend_radius_m)
    |   movel([0.639866, -1.466277, -2.511527, -0.734585, 1.570796, 2.210662],accel_mss,speed_ms,0,blend_radius_m)
    |   movel([0.640029, -1.467820, -2.510240, -0.734329, 1.570796, 2.210825],accel_mss,speed_ms,0,blend_radius_m)
    |   movel([0.640851, -1.470424, -2.508059, -0.733906, 1.570796, 2.211647],accel_mss,speed_ms,0,blend_radius_m)
    |   movel([0.641506, -1.471581, -2.507086, -0.733721, 1.570796, 2.212302],accel_mss,speed_ms,0,blend_radius_m)
    |   movel([0.642329, -1.472704, -2.506141, -0.733544, 1.570796, 2.213125],accel_mss,speed_ms,0,blend_radius_m)
    |   movel([0.642963, -1.473908, -2.505125, -0.733357, 1.570796, 2.213759],accel_mss,speed_ms,0,blend_radius_m)
    |   movel([0.643099, -1.474574, -2.504561, -0.733254, 1.570796, 2.213895],accel_mss,speed_ms,0,blend_radius_m)
    |   movel([0.643056, -1.475303, -2.503944, -0.733142, 1.570796, 2.213852],accel_mss,speed_ms,0,blend_radius_m)
    |   movel([0.642918, -1.475698, -2.503609, -0.733082, 1.570796, 2.213714],accel_mss,speed_ms,0,blend_radius_m)
    |   movel([0.642669, -1.476082, -2.503284, -0.733024, 1.570796, 2.213466],accel_mss,speed_ms,0,blend_radius_m)
    |   movel([0.642340, -1.476371, -2.503039, -0.732980, 1.570796, 2.213136],accel_mss,speed_ms,0,blend_radius_m)
    |   movel([0.641958, -1.476477, -2.502948, -0.732964, 1.570796, 2.212754],accel_mss,speed_ms,0,blend_radius_m)
    |   movel([0.641515, -1.476223, -2.503164, -0.733002, 1.570796, 2.212311],accel_mss,speed_ms,0,blend_radius_m)
    |   movel([0.640075, -1.474344, -2.504756, -0.733289, 1.570796, 2.210872],accel_mss,speed_ms,0,blend_radius_m)
    |   movel([0.638982, -1.472230, -2.506541, -0.733619, 1.570796, 2.209778],accel_mss,speed_ms,0,blend_radius_m)
    |   movel([0.638629, -1.472579, -2.506246, -0.733564, 1.570796, 2.209425],accel_mss,speed_ms,0,blend_radius_m)
    |   movel([0.638365, -1.472967, -2.505919, -0.733503, 1.570796, 2.209162],accel_mss,speed_ms,0,blend_radius_m)
    |   movel([0.638079, -1.473837, -2.505185, -0.733368, 1.570796, 2.208875],accel_mss,speed_ms,0,blend_radius_m)
    |   movel([0.638058, -1.474782, -2.504385, -0.733222, 1.570796, 2.208855],accel_mss,speed_ms,0,blend_radius_m)
    |   movel([0.638230, -1.475759, -2.503558, -0.733073, 1.570796, 2.209026],accel_mss,speed_ms,0,blend_radius_m)
    |   movel([0.638904, -1.477598, -2.501995, -0.732796, 1.570796, 2.209700],accel_mss,speed_ms,0,blend_radius_m)
    |   movel([0.639570, -1.478960, -2.500835, -0.732594, 1.570796, 2.210367],accel_mss,speed_ms,0,blend_radius_m)
    |   movel([0.639752, -1.479499, -2.500375, -0.732515, 1.570796, 2.210548],accel_mss,speed_ms,0,blend_radius_m)
    |   movel([0.639728, -1.479795, -2.500122, -0.732472, 1.570796, 2.210525],accel_mss,speed_ms,0,blend_radius_m)
    |   movel([0.639572, -1.480098, -2.499864, -0.732428, 1.570796, 2.210369],accel_mss,speed_ms,0,blend_radius_m)
    |   movel([0.639281, -1.480378, -2.499624, -0.732387, 1.570796, 2.210078],accel_mss,speed_ms,0,blend_radius_m)
    |   movel([0.638997, -1.480507, -2.499514, -0.732368, 1.570796, 2.209793],accel_mss,speed_ms,0,blend_radius_m)
    |   movel([0.638451, -1.480478, -2.499539, -0.732373, 1.570796, 2.209248],accel_mss,speed_ms,0,blend_radius_m)
    |   movel([0.637722, -1.480353, -2.499646, -0.732391, 1.570796, 2.208518],accel_mss,speed_ms,0,blend_radius_m)
    |   movel([0.637511, -1.480458, -2.499555, -0.732375, 1.570796, 2.208308],accel_mss,speed_ms,0,blend_radius_m)
    |   movel([0.637299, -1.480720, -2.499332, -0.732338, 1.570796, 2.208095],accel_mss,speed_ms,0,blend_radius_m)
    |   movel([0.637184, -1.481038, -2.499059, -0.732292, 1.570796, 2.207981],accel_mss,speed_ms,0,blend_radius_m)
    |   movel([0.637173, -1.481764, -2.498437, -0.732188, 1.570796, 2.207969],accel_mss,speed_ms,0,blend_radius_m)
    |   movel([0.637454, -1.483028, -2.497352, -0.732009, 1.570796, 2.208251],accel_mss,speed_ms,0,blend_radius_m)
    |   movel([0.639119, -1.488150, -2.492930, -0.731309, 1.570796, 2.209915],accel_mss,speed_ms,0,blend_radius_m)
    |   movel([0.639203, -1.488702, -2.492451, -0.731236, 1.570796, 2.209999],accel_mss,speed_ms,0,blend_radius_m)
    |   movel([0.639148, -1.489297, -2.491934, -0.731158, 1.570796, 2.209944],accel_mss,speed_ms,0,blend_radius_m)
    |   movel([0.638894, -1.489854, -2.491449, -0.731086, 1.570796, 2.209690],accel_mss,speed_ms,0,blend_radius_m)
    |   movel([0.638384, -1.490289, -2.491071, -0.731029, 1.570796, 2.209180],accel_mss,speed_ms,0,blend_radius_m)
    |   movel([0.637804, -1.490445, -2.490935, -0.731009, 1.570796, 2.208600],accel_mss,speed_ms,0,blend_radius_m)
    |   movel([0.637303, -1.490327, -2.491037, -0.731024, 1.570796, 2.208099],accel_mss,speed_ms,0,blend_radius_m)
    |   movel([0.636892, -1.490027, -2.491299, -0.731063, 1.570796, 2.207688],accel_mss,speed_ms,0,blend_radius_m)
    |   movel([0.636580, -1.489644, -2.491632, -0.731113, 1.570796, 2.207376],accel_mss,speed_ms,0,blend_radius_m)
    |   movel([0.635083, -1.487144, -2.493802, -0.731443, 1.570796, 2.205879],accel_mss,speed_ms,0,blend_radius_m)
    |   movel([0.633756, -1.484529, -2.496061, -0.731799, 1.570796, 2.204552],accel_mss,speed_ms,0,blend_radius_m)
    |   movel([0.632600, -1.481802, -2.498404, -0.732182, 1.570796, 2.203396],accel_mss,speed_ms,0,blend_radius_m)
    |   movel([0.631623, -1.478968, -2.500828, -0.732593, 1.570796, 2.202419],accel_mss,speed_ms,0,blend_radius_m)
    |   movel([0.631337, -1.477879, -2.501756, -0.732754, 1.570796, 2.202133],accel_mss,speed_ms,0,blend_radius_m)
    |   movel([0.631258, -1.476708, -2.502752, -0.732929, 1.570796, 2.202055],accel_mss,speed_ms,0,blend_radius_m)
    |   movel([0.631373, -1.475970, -2.503379, -0.733040, 1.570796, 2.202169],accel_mss,speed_ms,0,blend_radius_m)
    |   movel([0.631585, -1.475215, -2.504019, -0.733155, 1.570796, 2.202381],accel_mss,speed_ms,0,blend_radius_m)
    |   movel([0.632182, -1.473679, -2.505318, -0.733392, 1.570796, 2.202978],accel_mss,speed_ms,0,blend_radius_m)
    |   movel([0.634868, -1.468171, -2.509946, -0.734271, 1.570796, 2.205664],accel_mss,speed_ms,0,blend_radius_m)
    |   movel([0.635483, -1.466605, -2.511254, -0.734530, 1.570796, 2.206279],accel_mss,speed_ms,0,blend_radius_m)
    |   movel([0.635855, -1.465194, -2.512429, -0.734766, 1.570796, 2.206652],accel_mss,speed_ms,0,blend_radius_m)
    |   movel([0.635914, -1.464584, -2.512936, -0.734870, 1.570796, 2.206711],accel_mss,speed_ms,0,blend_radius_m)
    |   movel([0.635871, -1.464053, -2.513376, -0.734960, 1.570796, 2.206667],accel_mss,speed_ms,0,blend_radius_m)
    |   movel([0.635709, -1.463622, -2.513734, -0.735033, 1.570796, 2.206506],accel_mss,speed_ms,0,blend_radius_m)
    |   movel([0.635418, -1.463300, -2.514000, -0.735088, 1.570796, 2.206215],accel_mss,speed_ms,0,blend_radius_m)
    |   movel([0.634721, -1.462936, -2.514302, -0.735151, 1.570796, 2.205518],accel_mss,speed_ms,0,blend_radius_m)
    |   movel([0.634424, -1.462720, -2.514481, -0.735188, 1.570796, 2.205220],accel_mss,speed_ms,0,blend_radius_m)
    |   movel([0.634271, -1.462407, -2.514740, -0.735242, 1.570796, 2.205068],accel_mss,speed_ms,0,blend_radius_m)
    |   movel([0.634407, -1.461807, -2.515236, -0.735346, 1.570796, 2.205203],accel_mss,speed_ms,0,blend_radius_m)
    |   movel([0.634800, -1.461179, -2.515754, -0.735456, 1.570796, 2.205597],accel_mss,speed_ms,0,blend_radius_m)
    |   movel([0.636148, -1.459190, -2.517393, -0.735807, 1.570796, 2.206945],accel_mss,speed_ms,0,blend_radius_m)
    |   movel([0.637367, -1.457182, -2.519040, -0.736167, 1.570796, 2.208163],accel_mss,speed_ms,0,blend_radius_m)
    |   movel([0.639488, -1.453116, -2.522357, -0.736916, 1.570796, 2.210284],accel_mss,speed_ms,0,blend_radius_m)
    |   movel([0.641323, -1.448978, -2.525707, -0.737704, 1.570796, 2.212119],accel_mss,speed_ms,0,blend_radius_m)
    |   movel([0.643024, -1.444766, -2.529089, -0.738534, 1.570796, 2.213820],accel_mss,speed_ms,0,blend_radius_m)
    |   speed_ms = 0.005
    |   movel([0.643024, -1.436436, -2.525376, -0.750577, 1.570796, 2.213820],accel_mss,speed_ms,0,blend_radius_m)
    |   speed_ms = 0.040
    |   movel([0.637764, -1.442161, -2.520832, -0.749396, 1.570796, 2.208560],accel_mss,speed_ms,0,blend_radius_m)
    |   speed_ms = 0.005
    |   movel([0.637764, -1.450447, -2.524521, -0.737421, 1.570796, 2.208560],accel_mss,speed_ms,0,blend_radius_m)
    |   speed_ms = 0.025
    |   movel([0.634464, -1.454408, -2.521306, -0.736675, 1.570796, 2.205260],accel_mss,speed_ms,0,blend_radius_m)
    |   movel([0.632715, -1.456330, -2.519737, -0.736322, 1.570796, 2.203511],accel_mss,speed_ms,0,blend_radius_m)
    |   movel([0.630907, -1.458208, -2.518199, -0.735982, 1.570796, 2.201703],accel_mss,speed_ms,0,blend_radius_m)
    |   movel([0.630497, -1.456900, -2.519271, -0.736218, 1.570796, 2.201294],accel_mss,speed_ms,0,blend_radius_m)
    |   movel([0.630400, -1.456693, -2.519440, -0.736256, 1.570796, 2.201197],accel_mss,speed_ms,0,blend_radius_m)
    |   movel([0.630199, -1.456595, -2.519521, -0.736274, 1.570796, 2.200995],accel_mss,speed_ms,0,blend_radius_m)
    |   movel([0.629906, -1.456693, -2.519440, -0.736256, 1.570796, 2.200702],accel_mss,speed_ms,0,blend_radius_m)
    |   movel([0.629627, -1.456902, -2.519269, -0.736218, 1.570796, 2.200423],accel_mss,speed_ms,0,blend_radius_m)
    |   movel([0.627898, -1.458194, -2.518210, -0.735985, 1.570796, 2.198694],accel_mss,speed_ms,0,blend_radius_m)
    |   movel([0.626047, -1.459278, -2.517320, -0.735791, 1.570796, 2.196843],accel_mss,speed_ms,0,blend_radius_m)
    |   movel([0.625596, -1.459460, -2.517171, -0.735759, 1.570796, 2.196392],accel_mss,speed_ms,0,blend_radius_m)
    |   movel([0.625231, -1.459431, -2.517194, -0.735764, 1.570796, 2.196027],accel_mss,speed_ms,0,blend_radius_m)
    |   movel([0.625146, -1.459173, -2.517406, -0.735810, 1.570796, 2.195943],accel_mss,speed_ms,0,blend_radius_m)
    |   movel([0.625241, -1.458837, -2.517683, -0.735870, 1.570796, 2.196037],accel_mss,speed_ms,0,blend_radius_m)
    |   movel([0.626199, -1.456787, -2.519363, -0.736239, 1.570796, 2.196995],accel_mss,speed_ms,0,blend_radius_m)
    |   movel([0.627476, -1.454770, -2.521011, -0.736608, 1.570796, 2.198272],accel_mss,speed_ms,0,blend_radius_m)
    |   speed_ms = 0.005
    |   movel([0.627476, -1.446519, -2.517340, -0.748530, 1.570796, 2.198272],accel_mss,speed_ms,0,blend_radius_m)
    |   speed_ms = 0.040
    |   movel([0.627988, -1.451771, -2.513092, -0.747526, 1.570796, 2.198784],accel_mss,speed_ms,0,blend_radius_m)
    |   speed_ms = 0.005
    |   movel([0.627988, -1.459981, -2.516742, -0.735666, 1.570796, 2.198784],accel_mss,speed_ms,0,blend_radius_m)
    |   speed_ms = 0.025
    |   movel([0.626151, -1.462942, -2.514297, -0.735150, 1.570796, 2.196948],accel_mss,speed_ms,0,blend_radius_m)
    |   movel([0.625097, -1.464385, -2.513101, -0.734903, 1.570796, 2.195893],accel_mss,speed_ms,0,blend_radius_m)
    |   movel([0.622748, -1.467165, -2.510787, -0.734437, 1.570796, 2.193545],accel_mss,speed_ms,0,blend_radius_m)
    |   movel([0.621462, -1.468491, -2.509679, -0.734219, 1.570796, 2.192259],accel_mss,speed_ms,0,blend_radius_m)
    |   movel([0.618694, -1.470988, -2.507585, -0.733816, 1.570796, 2.189491],accel_mss,speed_ms,0,blend_radius_m)
    |   movel([0.619378, -1.470024, -2.508394, -0.733970, 1.570796, 2.190174],accel_mss,speed_ms,0,blend_radius_m)
    |   movel([0.619797, -1.469022, -2.509234, -0.734132, 1.570796, 2.190594],accel_mss,speed_ms,0,blend_radius_m)
    |   movel([0.619930, -1.468054, -2.510045, -0.734291, 1.570796, 2.190726],accel_mss,speed_ms,0,blend_radius_m)
    |   movel([0.619753, -1.467190, -2.510766, -0.734433, 1.570796, 2.190549],accel_mss,speed_ms,0,blend_radius_m)
    |   speed_ms = 0.005
    |   movel([0.619753, -1.459037, -2.507146, -0.746205, 1.570796, 2.190549],accel_mss,speed_ms,0,blend_radius_m)
    |   speed_ms = 0.040
    |   movel([0.608750, -1.458273, -2.507776, -0.746340, 1.570796, 2.179546],accel_mss,speed_ms,0,blend_radius_m)
    |   speed_ms = 0.005
    |   movel([0.608750, -1.466431, -2.511399, -0.734559, 1.570796, 2.179546],accel_mss,speed_ms,0,blend_radius_m)
    |   speed_ms = 0.025
    |   movel([0.606276, -1.467605, -2.510420, -0.734364, 1.570796, 2.177072],accel_mss,speed_ms,0,blend_radius_m)
    |   movel([0.603766, -1.468519, -2.509656, -0.734215, 1.570796, 2.174563],accel_mss,speed_ms,0,blend_radius_m)
    |   movel([0.601263, -1.469162, -2.509117, -0.734110, 1.570796, 2.172059],accel_mss,speed_ms,0,blend_radius_m)
    |   movel([0.598809, -1.469521, -2.508816, -0.734051, 1.570796, 2.169605],accel_mss,speed_ms,0,blend_radius_m)
    |   movel([0.599716, -1.468751, -2.509462, -0.734177, 1.570796, 2.170512],accel_mss,speed_ms,0,blend_radius_m)
    |   movel([0.600486, -1.467955, -2.510127, -0.734307, 1.570796, 2.171283],accel_mss,speed_ms,0,blend_radius_m)
    |   movel([0.601057, -1.467211, -2.510748, -0.734429, 1.570796, 2.171853],accel_mss,speed_ms,0,blend_radius_m)
    |   movel([0.601366, -1.466593, -2.511264, -0.734532, 1.570796, 2.172162],accel_mss,speed_ms,0,blend_radius_m)
    |   movel([0.601345, -1.466181, -2.511607, -0.734601, 1.570796, 2.172142],accel_mss,speed_ms,0,blend_radius_m)
    |   movel([0.601194, -1.466075, -2.511695, -0.734618, 1.570796, 2.171990],accel_mss,speed_ms,0,blend_radius_m)
    |   movel([0.600934, -1.466048, -2.511718, -0.734623, 1.570796, 2.171730],accel_mss,speed_ms,0,blend_radius_m)
    |   movel([0.600067, -1.466274, -2.511529, -0.734585, 1.570796, 2.170864],accel_mss,speed_ms,0,blend_radius_m)
    |   movel([0.597596, -1.467480, -2.510524, -0.734385, 1.570796, 2.168392],accel_mss,speed_ms,0,blend_radius_m)
    |   movel([0.596477, -1.467956, -2.510126, -0.734307, 1.570796, 2.167273],accel_mss,speed_ms,0,blend_radius_m)
    |   movel([0.594203, -1.468674, -2.509526, -0.734189, 1.570796, 2.164999],accel_mss,speed_ms,0,blend_radius_m)
    |   movel([0.593077, -1.468905, -2.509333, -0.734152, 1.570796, 2.163873],accel_mss,speed_ms,0,blend_radius_m)
    |   movel([0.591978, -1.469037, -2.509222, -0.734130, 1.570796, 2.162775],accel_mss,speed_ms,0,blend_radius_m)
    |   movel([0.590919, -1.469071, -2.509194, -0.734125, 1.570796, 2.161716],accel_mss,speed_ms,0,blend_radius_m)
    |   movel([0.589919, -1.468994, -2.509258, -0.734137, 1.570796, 2.160715],accel_mss,speed_ms,0,blend_radius_m)
    |   movel([0.591630, -1.468026, -2.510068, -0.734295, 1.570796, 2.162426],accel_mss,speed_ms,0,blend_radius_m)
    |   movel([0.593324, -1.467014, -2.510913, -0.734462, 1.570796, 2.164121],accel_mss,speed_ms,0,blend_radius_m)
    |   movel([0.594264, -1.466177, -2.511611, -0.734601, 1.570796, 2.165060],accel_mss,speed_ms,0,blend_radius_m)
    |   movel([0.595003, -1.465226, -2.512402, -0.734761, 1.570796, 2.165799],accel_mss,speed_ms,0,blend_radius_m)
    |   movel([0.595149, -1.464828, -2.512733, -0.734828, 1.570796, 2.165945],accel_mss,speed_ms,0,blend_radius_m)
    |   movel([0.595062, -1.464545, -2.512968, -0.734876, 1.570796, 2.165858],accel_mss,speed_ms,0,blend_radius_m)
    |   movel([0.594686, -1.464428, -2.513065, -0.734896, 1.570796, 2.165483],accel_mss,speed_ms,0,blend_radius_m)
    |   movel([0.593960, -1.464526, -2.512983, -0.734879, 1.570796, 2.164756],accel_mss,speed_ms,0,blend_radius_m)
    |   movel([0.589880, -1.465593, -2.512097, -0.734699, 1.570796, 2.160677],accel_mss,speed_ms,0,blend_radius_m)
    |   movel([0.587928, -1.465897, -2.511843, -0.734648, 1.570796, 2.158724],accel_mss,speed_ms,0,blend_radius_m)
    |   movel([0.587015, -1.465903, -2.511839, -0.734647, 1.570796, 2.157811],accel_mss,speed_ms,0,blend_radius_m)
    |   movel([0.586157, -1.465776, -2.511945, -0.734669, 1.570796, 2.156953],accel_mss,speed_ms,0,blend_radius_m)
    |   speed_ms = 0.005
    |   movel([0.586157, -1.457612, -2.508319, -0.746458, 1.570796, 2.156953],accel_mss,speed_ms,0,blend_radius_m)
    |   speed_ms = 0.040
    |   movel([0.608445, -1.444545, -2.518925, -0.748919, 1.570796, 2.179242],accel_mss,speed_ms,0,blend_radius_m)
    |   speed_ms = 0.005
    |   movel([0.608445, -1.452812, -2.522604, -0.736973, 1.570796, 2.179242],accel_mss,speed_ms,0,blend_radius_m)
    |   speed_ms = 0.025
    |   movel([0.609102, -1.451455, -2.523704, -0.737229, 1.570796, 2.179898],accel_mss,speed_ms,0,blend_radius_m)
    |   movel([0.610004, -1.450153, -2.524759, -0.737478, 1.570796, 2.180800],accel_mss,speed_ms,0,blend_radius_m)
    |   movel([0.611115, -1.448916, -2.525757, -0.737716, 1.570796, 2.181912],accel_mss,speed_ms,0,blend_radius_m)
    |   movel([0.612394, -1.447766, -2.526683, -0.737940, 1.570796, 2.183190],accel_mss,speed_ms,0,blend_radius_m)
    |   movel([0.613809, -1.446716, -2.527526, -0.738146, 1.570796, 2.184605],accel_mss,speed_ms,0,blend_radius_m)
    |   movel([0.615315, -1.445789, -2.528270, -0.738330, 1.570796, 2.186111],accel_mss,speed_ms,0,blend_radius_m)
    |   movel([0.616882, -1.444997, -2.528905, -0.738488, 1.570796, 2.187678],accel_mss,speed_ms,0,blend_radius_m)
    |   movel([0.618464, -1.444359, -2.529414, -0.738615, 1.570796, 2.189261],accel_mss,speed_ms,0,blend_radius_m)
    |   movel([0.620408, -1.443761, -2.529892, -0.738736, 1.570796, 2.191205],accel_mss,speed_ms,0,blend_radius_m)
    |   movel([0.624291, -1.442705, -2.530734, -0.738950, 1.570796, 2.195087],accel_mss,speed_ms,0,blend_radius_m)
    |   movel([0.626231, -1.442020, -2.531280, -0.739089, 1.570796, 2.197028],accel_mss,speed_ms,0,blend_radius_m)
    |   movel([0.628170, -1.441040, -2.532058, -0.739290, 1.570796, 2.198966],accel_mss,speed_ms,0,blend_radius_m)
    |   movel([0.629096, -1.440430, -2.532542, -0.739416, 1.570796, 2.199893],accel_mss,speed_ms,0,blend_radius_m)
    |   movel([0.629958, -1.439753, -2.533079, -0.739557, 1.570796, 2.200754],accel_mss,speed_ms,0,blend_radius_m)
    |   movel([0.630728, -1.439017, -2.533662, -0.739710, 1.570796, 2.201524],accel_mss,speed_ms,0,blend_radius_m)
    |   movel([0.631381, -1.438234, -2.534281, -0.739874, 1.570796, 2.202177],accel_mss,speed_ms,0,blend_radius_m)
    |   movel([0.631884, -1.437414, -2.534928, -0.740047, 1.570796, 2.202680],accel_mss,speed_ms,0,blend_radius_m)
    |   movel([0.632210, -1.436568, -2.535594, -0.740227, 1.570796, 2.203006],accel_mss,speed_ms,0,blend_radius_m)
    |   speed_ms = 0.005
    |   movel([0.632210, -1.428174, -2.531847, -0.752368, 1.570796, 2.203006],accel_mss,speed_ms,0,blend_radius_m)
    |   speed_ms = 0.040
    |   movel([0.634472, -1.421241, -2.537198, -0.753950, 1.570796, 2.205268],accel_mss,speed_ms,0,blend_radius_m)
    |   speed_ms = 0.005
    |   movel([0.634472, -1.429688, -2.540974, -0.741726, 1.570796, 2.205268],accel_mss,speed_ms,0,blend_radius_m)
    |   speed_ms = 0.025
    |   movel([0.630966, -1.434319, -2.537361, -0.740709, 1.570796, 2.201762],accel_mss,speed_ms,0,blend_radius_m)
    |   movel([0.630012, -1.435247, -2.536633, -0.740509, 1.570796, 2.200808],accel_mss,speed_ms,0,blend_radius_m)
    |   movel([0.628877, -1.435944, -2.536085, -0.740360, 1.570796, 2.199673],accel_mss,speed_ms,0,blend_radius_m)
    |   movel([0.627663, -1.436404, -2.535723, -0.740262, 1.570796, 2.198460],accel_mss,speed_ms,0,blend_radius_m)
    |   movel([0.623784, -1.437426, -2.534919, -0.740045, 1.570796, 2.194581],accel_mss,speed_ms,0,blend_radius_m)
    |   movel([0.622396, -1.437944, -2.534510, -0.739935, 1.570796, 2.193193],accel_mss,speed_ms,0,blend_radius_m)
    |   movel([0.621022, -1.438571, -2.534015, -0.739804, 1.570796, 2.191818],accel_mss,speed_ms,0,blend_radius_m)
    |   movel([0.619676, -1.439294, -2.533443, -0.739652, 1.570796, 2.190472],accel_mss,speed_ms,0,blend_radius_m)
    |   movel([0.618436, -1.440141, -2.532772, -0.739476, 1.570796, 2.189232],accel_mss,speed_ms,0,blend_radius_m)
    |   movel([0.617280, -1.441094, -2.532016, -0.739279, 1.570796, 2.188076],accel_mss,speed_ms,0,blend_radius_m)
    |   movel([0.616136, -1.442049, -2.531256, -0.739083, 1.570796, 2.186932],accel_mss,speed_ms,0,blend_radius_m)
    |   movel([0.614930, -1.442905, -2.530575, -0.738909, 1.570796, 2.185726],accel_mss,speed_ms,0,blend_radius_m)
    |   movel([0.615593, -1.439744, -2.533086, -0.739559, 1.570796, 2.186390],accel_mss,speed_ms,0,blend_radius_m)
    |   movel([0.616059, -1.438916, -2.533742, -0.739731, 1.570796, 2.186855],accel_mss,speed_ms,0,blend_radius_m)
    |   movel([0.616636, -1.438140, -2.534355, -0.739894, 1.570796, 2.187432],accel_mss,speed_ms,0,blend_radius_m)
    |   movel([0.617323, -1.437413, -2.534928, -0.740047, 1.570796, 2.188119],accel_mss,speed_ms,0,blend_radius_m)
    |   movel([0.618129, -1.436734, -2.535464, -0.740191, 1.570796, 2.188926],accel_mss,speed_ms,0,blend_radius_m)
    |   movel([0.619413, -1.435981, -2.536056, -0.740352, 1.570796, 2.190209],accel_mss,speed_ms,0,blend_radius_m)
    |   movel([0.621123, -1.435253, -2.536628, -0.740508, 1.570796, 2.191920],accel_mss,speed_ms,0,blend_radius_m)
    |   movel([0.625153, -1.433842, -2.537735, -0.740812, 1.570796, 2.195949],accel_mss,speed_ms,0,blend_radius_m)
    |   movel([0.627133, -1.433147, -2.538278, -0.740963, 1.570796, 2.197930],accel_mss,speed_ms,0,blend_radius_m)
    |   movel([0.628867, -1.432445, -2.538827, -0.741117, 1.570796, 2.199663],accel_mss,speed_ms,0,blend_radius_m)
    |   movel([0.630181, -1.431732, -2.539383, -0.741273, 1.570796, 2.200977],accel_mss,speed_ms,0,blend_radius_m)
    |   movel([0.630630, -1.431367, -2.539668, -0.741354, 1.570796, 2.201426],accel_mss,speed_ms,0,blend_radius_m)
    |   movel([0.630911, -1.430993, -2.539959, -0.741436, 1.570796, 2.201707],accel_mss,speed_ms,0,blend_radius_m)
    |   speed_ms = 0.005
    |   movel([0.630911, -1.422556, -2.536188, -0.753645, 1.570796, 2.201707],accel_mss,speed_ms,0,blend_radius_m)
    |   speed_ms = 0.040
    |   movel([0.626406, -1.418603, -2.539215, -0.754571, 1.570796, 2.197203],accel_mss,speed_ms,0,blend_radius_m)
    |   speed_ms = 0.005
    |   movel([0.626406, -1.427071, -2.543002, -0.742316, 1.570796, 2.197203],accel_mss,speed_ms,0,blend_radius_m)
    |   speed_ms = 0.025
    |   movel([0.625978, -1.426676, -2.543308, -0.742406, 1.570796, 2.196775],accel_mss,speed_ms,0,blend_radius_m)
    |   movel([0.625701, -1.426178, -2.543692, -0.742519, 1.570796, 2.196497],accel_mss,speed_ms,0,blend_radius_m)
    |   movel([0.625515, -1.424957, -2.544632, -0.742799, 1.570796, 2.196311],accel_mss,speed_ms,0,blend_radius_m)
    |   movel([0.625692, -1.423549, -2.545715, -0.743125, 1.570796, 2.196488],accel_mss,speed_ms,0,blend_radius_m)
    |   movel([0.626077, -1.422092, -2.546832, -0.743466, 1.570796, 2.196873],accel_mss,speed_ms,0,blend_radius_m)
    |   movel([0.626302, -1.421561, -2.547237, -0.743590, 1.570796, 2.197098],accel_mss,speed_ms,0,blend_radius_m)
    |   movel([0.627024, -1.420869, -2.547766, -0.743754, 1.570796, 2.197820],accel_mss,speed_ms,0,blend_radius_m)
    |   movel([0.629266, -1.419088, -2.549123, -0.744177, 1.570796, 2.200063],accel_mss,speed_ms,0,blend_radius_m)
    |   movel([0.633612, -1.415346, -2.551960, -0.745083, 1.570796, 2.204409],accel_mss,speed_ms,0,blend_radius_m)
    |   movel([0.635707, -1.413393, -2.553432, -0.745564, 1.570796, 2.206503],accel_mss,speed_ms,0,blend_radius_m)
    |   speed_ms = 0.005
    |   movel([0.635707, -1.404821, -2.549586, -0.757982, 1.570796, 2.206503],accel_mss,speed_ms,0,blend_radius_m)
    |   speed_ms = 0.040
    |   movel([0.631730, -1.404605, -2.549746, -0.758038, 1.570796, 2.202526],accel_mss,speed_ms,0,blend_radius_m)
    |   speed_ms = 0.005
    |   movel([0.631730, -1.413178, -2.553593, -0.745617, 1.570796, 2.202526],accel_mss,speed_ms,0,blend_radius_m)
    |   speed_ms = 0.025
    |   movel([0.630561, -1.414434, -2.552648, -0.745307, 1.570796, 2.201357],accel_mss,speed_ms,0,blend_radius_m)
    |   movel([0.629275, -1.415602, -2.551767, -0.745021, 1.570796, 2.200071],accel_mss,speed_ms,0,blend_radius_m)
    |   movel([0.627884, -1.416569, -2.551035, -0.744785, 1.570796, 2.198680],accel_mss,speed_ms,0,blend_radius_m)
    |   movel([0.627150, -1.416945, -2.550750, -0.744694, 1.570796, 2.197947],accel_mss,speed_ms,0,blend_radius_m)
    |   movel([0.625657, -1.417523, -2.550312, -0.744554, 1.570796, 2.196453],accel_mss,speed_ms,0,blend_radius_m)
    |   movel([0.625143, -1.417996, -2.549953, -0.744440, 1.570796, 2.195940],accel_mss,speed_ms,0,blend_radius_m)
    |   movel([0.621578, -1.421930, -2.546956, -0.743504, 1.570796, 2.192374],accel_mss,speed_ms,0,blend_radius_m)
    |   movel([0.621243, -1.422316, -2.546660, -0.743413, 1.570796, 2.192039],accel_mss,speed_ms,0,blend_radius_m)
    |   movel([0.621016, -1.422721, -2.546349, -0.743318, 1.570796, 2.191812],accel_mss,speed_ms,0,blend_radius_m)
    |   movel([0.621038, -1.423264, -2.545933, -0.743192, 1.570796, 2.191834],accel_mss,speed_ms,0,blend_radius_m)
    |   movel([0.621320, -1.423696, -2.545602, -0.743091, 1.570796, 2.192117],accel_mss,speed_ms,0,blend_radius_m)
    |   movel([0.622190, -1.424884, -2.544689, -0.742816, 1.570796, 2.192987],accel_mss,speed_ms,0,blend_radius_m)
    |   movel([0.622880, -1.426189, -2.543683, -0.742517, 1.570796, 2.193677],accel_mss,speed_ms,0,blend_radius_m)
    |   movel([0.623286, -1.427633, -2.542568, -0.742188, 1.570796, 2.194082],accel_mss,speed_ms,0,blend_radius_m)
    |   movel([0.623292, -1.429238, -2.541324, -0.741827, 1.570796, 2.194088],accel_mss,speed_ms,0,blend_radius_m)
    |   speed_ms = 0.005
    |   movel([0.623292, -1.420787, -2.537546, -0.754056, 1.570796, 2.194088],accel_mss,speed_ms,0,blend_radius_m)
    |   speed_ms = 0.040
    |   movel([0.614239, -1.430940, -2.529692, -0.751757, 1.570796, 2.185036],accel_mss,speed_ms,0,blend_radius_m)
    |   speed_ms = 0.005
    |   movel([0.614239, -1.439312, -2.533428, -0.739649, 1.570796, 2.185036],accel_mss,speed_ms,0,blend_radius_m)
    |   speed_ms = 0.025
    |   movel([0.613899, -1.439397, -2.533361, -0.739631, 1.570796, 2.184695],accel_mss,speed_ms,0,blend_radius_m)
    |   movel([0.613539, -1.439584, -2.533213, -0.739592, 1.570796, 2.184336],accel_mss,speed_ms,0,blend_radius_m)
    |   movel([0.611897, -1.440794, -2.532254, -0.739341, 1.570796, 2.182693],accel_mss,speed_ms,0,blend_radius_m)
    |   movel([0.611689, -1.440847, -2.532211, -0.739330, 1.570796, 2.182486],accel_mss,speed_ms,0,blend_radius_m)
    |   movel([0.611472, -1.440734, -2.532301, -0.739353, 1.570796, 2.182269],accel_mss,speed_ms,0,blend_radius_m)
    |   movel([0.611391, -1.440464, -2.532516, -0.739409, 1.570796, 2.182188],accel_mss,speed_ms,0,blend_radius_m)
    |   movel([0.611527, -1.439641, -2.533168, -0.739580, 1.570796, 2.182323],accel_mss,speed_ms,0,blend_radius_m)
    |   movel([0.612164, -1.438124, -2.534368, -0.739897, 1.570796, 2.182960],accel_mss,speed_ms,0,blend_radius_m)
    |   movel([0.613130, -1.436783, -2.535425, -0.740181, 1.570796, 2.183926],accel_mss,speed_ms,0,blend_radius_m)
    |   movel([0.614280, -1.435499, -2.536435, -0.740455, 1.570796, 2.185077],accel_mss,speed_ms,0,blend_radius_m)
    |   movel([0.615503, -1.434287, -2.537386, -0.740716, 1.570796, 2.186300],accel_mss,speed_ms,0,blend_radius_m)
    |   movel([0.616788, -1.433202, -2.538236, -0.740951, 1.570796, 2.187584],accel_mss,speed_ms,0,blend_radius_m)
    |   movel([0.618128, -1.432240, -2.538987, -0.741162, 1.570796, 2.188924],accel_mss,speed_ms,0,blend_radius_m)
    |   movel([0.619521, -1.431398, -2.539644, -0.741347, 1.570796, 2.190317],accel_mss,speed_ms,0,blend_radius_m)
    |   movel([0.620965, -1.430671, -2.540210, -0.741508, 1.570796, 2.191761],accel_mss,speed_ms,0,blend_radius_m)
    |   movel([0.622453, -1.430055, -2.540689, -0.741644, 1.570796, 2.193249],accel_mss,speed_ms,0,blend_radius_m)
    |   movel([0.623986, -1.429546, -2.541085, -0.741758, 1.570796, 2.194782],accel_mss,speed_ms,0,blend_radius_m)
    |   movel([0.625558, -1.429138, -2.541401, -0.741849, 1.570796, 2.196355],accel_mss,speed_ms,0,blend_radius_m)
    |   movel([0.627800, -1.428405, -2.541970, -0.742014, 1.570796, 2.198597],accel_mss,speed_ms,0,blend_radius_m)
    |   movel([0.630263, -1.427347, -2.542789, -0.742253, 1.570796, 2.201059],accel_mss,speed_ms,0,blend_radius_m)
    |   movel([0.632999, -1.425997, -2.543831, -0.742561, 1.570796, 2.203795],accel_mss,speed_ms,0,blend_radius_m)
    |   speed_ms = 0.005
    |   movel([0.632999, -1.417521, -2.540039, -0.754829, 1.570796, 2.203795],accel_mss,speed_ms,0,blend_radius_m)
    |   speed_ms = 0.040
    |   movel([0.631529, -1.416683, -2.540677, -0.755030, 1.570796, 2.202326],accel_mss,speed_ms,0,blend_radius_m)
    |   speed_ms = 0.005
    |   movel([0.631529, -1.425165, -2.544473, -0.742752, 1.570796, 2.202326],accel_mss,speed_ms,0,blend_radius_m)
    |   speed_ms = 0.025
    |   movel([0.634472, -1.422332, -2.546648, -0.743409, 1.570796, 2.205269],accel_mss,speed_ms,0,blend_radius_m)
    |   movel([0.637560, -1.419600, -2.548734, -0.744055, 1.570796, 2.208356],accel_mss,speed_ms,0,blend_radius_m)
    |   movel([0.639176, -1.418327, -2.549702, -0.744360, 1.570796, 2.209972],accel_mss,speed_ms,0,blend_radius_m)
    |   movel([0.640843, -1.417142, -2.550601, -0.744646, 1.570796, 2.211640],accel_mss,speed_ms,0,blend_radius_m)
    |   movel([0.642574, -1.416069, -2.551413, -0.744907, 1.570796, 2.213371],accel_mss,speed_ms,0,blend_radius_m)
    |   movel([0.644367, -1.415131, -2.552122, -0.745136, 1.570796, 2.215163],accel_mss,speed_ms,0,blend_radius_m)
    |   movel([0.649060, -1.413130, -2.553629, -0.745629, 1.570796, 2.219856],accel_mss,speed_ms,0,blend_radius_m)
    |   movel([0.651133, -1.412130, -2.554381, -0.745878, 1.570796, 2.221930],accel_mss,speed_ms,0,blend_radius_m)
    |   movel([0.652150, -1.411557, -2.554810, -0.746021, 1.570796, 2.222947],accel_mss,speed_ms,0,blend_radius_m)
    |   movel([0.653131, -1.410897, -2.555305, -0.746187, 1.570796, 2.223928],accel_mss,speed_ms,0,blend_radius_m)
    |   movel([0.655731, -1.408453, -2.557129, -0.746806, 1.570796, 2.226527],accel_mss,speed_ms,0,blend_radius_m)
    |   speed_ms = 0.005
    |   movel([0.655731, -1.399844, -2.553262, -0.759283, 1.570796, 2.226527],accel_mss,speed_ms,0,blend_radius_m)
    |   speed_ms = 0.040
    |   movel([0.661836, -1.394252, -2.557350, -0.760788, 1.570796, 2.232632],accel_mss,speed_ms,0,blend_radius_m)
    |   speed_ms = 0.005
    |   movel([0.661836, -1.402902, -2.561241, -0.748245, 1.570796, 2.232632],accel_mss,speed_ms,0,blend_radius_m)
    |   speed_ms = 0.025
    |   movel([0.663890, -1.400838, -2.562759, -0.748792, 1.570796, 2.234687],accel_mss,speed_ms,0,blend_radius_m)
    |   movel([0.665035, -1.399965, -2.563398, -0.749025, 1.570796, 2.235831],accel_mss,speed_ms,0,blend_radius_m)
    |   movel([0.666278, -1.399312, -2.563877, -0.749200, 1.570796, 2.237075],accel_mss,speed_ms,0,blend_radius_m)
    |   movel([0.667177, -1.399037, -2.564078, -0.749274, 1.570796, 2.237974],accel_mss,speed_ms,0,blend_radius_m)
    |   movel([0.668058, -1.398894, -2.564182, -0.749313, 1.570796, 2.238854],accel_mss,speed_ms,0,blend_radius_m)
    |   movel([0.669780, -1.398801, -2.564250, -0.749338, 1.570796, 2.240576],accel_mss,speed_ms,0,blend_radius_m)
    |   movel([0.671376, -1.398578, -2.564413, -0.749398, 1.570796, 2.242173],accel_mss,speed_ms,0,blend_radius_m)
    |   movel([0.672788, -1.398079, -2.564777, -0.749533, 1.570796, 2.243584],accel_mss,speed_ms,0,blend_radius_m)
    |   movel([0.675757, -1.396456, -2.565959, -0.749974, 1.570796, 2.246553],accel_mss,speed_ms,0,blend_radius_m)
    |   movel([0.676370, -1.396174, -2.566165, -0.750051, 1.570796, 2.247166],accel_mss,speed_ms,0,blend_radius_m)
    |   movel([0.676978, -1.396006, -2.566287, -0.750097, 1.570796, 2.247775],accel_mss,speed_ms,0,blend_radius_m)
    |   movel([0.678181, -1.395918, -2.566350, -0.750121, 1.570796, 2.248978],accel_mss,speed_ms,0,blend_radius_m)
    |   movel([0.680510, -1.396020, -2.566276, -0.750093, 1.570796, 2.251307],accel_mss,speed_ms,0,blend_radius_m)
    |   movel([0.683082, -1.395846, -2.566403, -0.750140, 1.570796, 2.253879],accel_mss,speed_ms,0,blend_radius_m)
    |   movel([0.684409, -1.395623, -2.566565, -0.750202, 1.570796, 2.255205],accel_mss,speed_ms,0,blend_radius_m)
    |   movel([0.685767, -1.395218, -2.566859, -0.750313, 1.570796, 2.256564],accel_mss,speed_ms,0,blend_radius_m)
    |   movel([0.686865, -1.394669, -2.567256, -0.750464, 1.570796, 2.257661],accel_mss,speed_ms,0,blend_radius_m)
    |   movel([0.687861, -1.393908, -2.567807, -0.750674, 1.570796, 2.258657],accel_mss,speed_ms,0,blend_radius_m)
    |   movel([0.688550, -1.393039, -2.568435, -0.750915, 1.570796, 2.259346],accel_mss,speed_ms,0,blend_radius_m)
    |   movel([0.688714, -1.392599, -2.568753, -0.751037, 1.570796, 2.259510],accel_mss,speed_ms,0,blend_radius_m)
    |   movel([0.688723, -1.392174, -2.569060, -0.751156, 1.570796, 2.259519],accel_mss,speed_ms,0,blend_radius_m)
    |   movel([0.688416, -1.391422, -2.569601, -0.751366, 1.570796, 2.259212],accel_mss,speed_ms,0,blend_radius_m)
    |   movel([0.687831, -1.390766, -2.570073, -0.751550, 1.570796, 2.258627],accel_mss,speed_ms,0,blend_radius_m)
    |   movel([0.687019, -1.390220, -2.570465, -0.751704, 1.570796, 2.257815],accel_mss,speed_ms,0,blend_radius_m)
    |   movel([0.686046, -1.389794, -2.570771, -0.751824, 1.570796, 2.256842],accel_mss,speed_ms,0,blend_radius_m)
    |   movel([0.684965, -1.389510, -2.570975, -0.751904, 1.570796, 2.255761],accel_mss,speed_ms,0,blend_radius_m)
    |   movel([0.683839, -1.389375, -2.571072, -0.751943, 1.570796, 2.254635],accel_mss,speed_ms,0,blend_radius_m)
    |   movel([0.682724, -1.389408, -2.571048, -0.751933, 1.570796, 2.253520],accel_mss,speed_ms,0,blend_radius_m)
    |   movel([0.681679, -1.389620, -2.570896, -0.751873, 1.570796, 2.252475],accel_mss,speed_ms,0,blend_radius_m)
    |   movel([0.680107, -1.390284, -2.570419, -0.751686, 1.570796, 2.250903],accel_mss,speed_ms,0,blend_radius_m)
    |   movel([0.675473, -1.392714, -2.568670, -0.751005, 1.570796, 2.246269],accel_mss,speed_ms,0,blend_radius_m)
    |   movel([0.672351, -1.394092, -2.567674, -0.750623, 1.570796, 2.243147],accel_mss,speed_ms,0,blend_radius_m)
    |   movel([0.669641, -1.394935, -2.567064, -0.750390, 1.570796, 2.240437],accel_mss,speed_ms,0,blend_radius_m)
    |   movel([0.668305, -1.395322, -2.566783, -0.750284, 1.570796, 2.239101],accel_mss,speed_ms,0,blend_radius_m)
    |   movel([0.666980, -1.395830, -2.566414, -0.750145, 1.570796, 2.237776],accel_mss,speed_ms,0,blend_radius_m)
    |   movel([0.665633, -1.396532, -2.565904, -0.749953, 1.570796, 2.236430],accel_mss,speed_ms,0,blend_radius_m)
    |   movel([0.664346, -1.397350, -2.565309, -0.749730, 1.570796, 2.235142],accel_mss,speed_ms,0,blend_radius_m)
    |   movel([0.663112, -1.398265, -2.564641, -0.749482, 1.570796, 2.233909],accel_mss,speed_ms,0,blend_radius_m)
    |   movel([0.661932, -1.399254, -2.563919, -0.749216, 1.570796, 2.232728],accel_mss,speed_ms,0,blend_radius_m)
    |   movel([0.659712, -1.401374, -2.562365, -0.748649, 1.570796, 2.230508],accel_mss,speed_ms,0,blend_radius_m)
    |   movel([0.657647, -1.403546, -2.560767, -0.748076, 1.570796, 2.228444],accel_mss,speed_ms,0,blend_radius_m)
    |   speed_ms = 0.005
    |   movel([0.657647, -1.394900, -2.556878, -0.760611, 1.570796, 2.228444],accel_mss,speed_ms,0,blend_radius_m)
    |   speed_ms = 0.040
    |   movel([0.654415, -1.395213, -2.556651, -0.760526, 1.570796, 2.225212],accel_mss,speed_ms,0,blend_radius_m)
    |   speed_ms = 0.005
    |   movel([0.654415, -1.403856, -2.560538, -0.747995, 1.570796, 2.225212],accel_mss,speed_ms,0,blend_radius_m)
    |   speed_ms = 0.025
    |   movel([0.657764, -1.400491, -2.563013, -0.748885, 1.570796, 2.228560],accel_mss,speed_ms,0,blend_radius_m)
    |   movel([0.659213, -1.399123, -2.564014, -0.749251, 1.570796, 2.230010],accel_mss,speed_ms,0,blend_radius_m)
    |   movel([0.660598, -1.397708, -2.565048, -0.749633, 1.570796, 2.231394],accel_mss,speed_ms,0,blend_radius_m)
    |   movel([0.661658, -1.396409, -2.565994, -0.749987, 1.570796, 2.232454],accel_mss,speed_ms,0,blend_radius_m)
    |   movel([0.662556, -1.395052, -2.566979, -0.750358, 1.570796, 2.233353],accel_mss,speed_ms,0,blend_radius_m)
    |   movel([0.663277, -1.393664, -2.567984, -0.750741, 1.570796, 2.234073],accel_mss,speed_ms,0,blend_radius_m)
    |   movel([0.663803, -1.392274, -2.568987, -0.751128, 1.570796, 2.234600],accel_mss,speed_ms,0,blend_radius_m)
    |   movel([0.664421, -1.392300, -2.568969, -0.751120, 1.570796, 2.235217],accel_mss,speed_ms,0,blend_radius_m)
    |   movel([0.664952, -1.392477, -2.568841, -0.751071, 1.570796, 2.235749],accel_mss,speed_ms,0,blend_radius_m)
    |   movel([0.665902, -1.393010, -2.568456, -0.750923, 1.570796, 2.236698],accel_mss,speed_ms,0,blend_radius_m)
    |   movel([0.666957, -1.393447, -2.568141, -0.750801, 1.570796, 2.237753],accel_mss,speed_ms,0,blend_radius_m)
    |   movel([0.667567, -1.393492, -2.568108, -0.750789, 1.570796, 2.238364],accel_mss,speed_ms,0,blend_radius_m)
    |   movel([0.668235, -1.393324, -2.568229, -0.750835, 1.570796, 2.239032],accel_mss,speed_ms,0,blend_radius_m)
    |   movel([0.676287, -1.390042, -2.570593, -0.751754, 1.570796, 2.247083],accel_mss,speed_ms,0,blend_radius_m)
    |   movel([0.676745, -1.389077, -2.571285, -0.752027, 1.570796, 2.247541],accel_mss,speed_ms,0,blend_radius_m)
    |   movel([0.676931, -1.388102, -2.571983, -0.752304, 1.570796, 2.247728],accel_mss,speed_ms,0,blend_radius_m)
    |   movel([0.676838, -1.387168, -2.572650, -0.752571, 1.570796, 2.247634],accel_mss,speed_ms,0,blend_radius_m)
    |   movel([0.676462, -1.386329, -2.573248, -0.752812, 1.570796, 2.247259],accel_mss,speed_ms,0,blend_radius_m)
    |   movel([0.677727, -1.386688, -2.572992, -0.752709, 1.570796, 2.248523],accel_mss,speed_ms,0,blend_radius_m)
    |   movel([0.678785, -1.387289, -2.572563, -0.752536, 1.570796, 2.249582],accel_mss,speed_ms,0,blend_radius_m)
    |   movel([0.679587, -1.388095, -2.571987, -0.752306, 1.570796, 2.250383],accel_mss,speed_ms,0,blend_radius_m)
    |   movel([0.680086, -1.389070, -2.571290, -0.752029, 1.570796, 2.250882],accel_mss,speed_ms,0,blend_radius_m)
    |   speed_ms = 0.005
    |   movel([0.680086, -1.380317, -2.567338, -0.764734, 1.570796, 2.250882],accel_mss,speed_ms,0,blend_radius_m)
    |   speed_ms = 0.040
    |   movel([0.682625, -1.376904, -2.569742, -0.765743, 1.570796, 2.253421],accel_mss,speed_ms,0,blend_radius_m)
    |   speed_ms = 0.005
    |   movel([0.682625, -1.385682, -2.573709, -0.752998, 1.570796, 2.253421],accel_mss,speed_ms,0,blend_radius_m)
    |   speed_ms = 0.025
    |   movel([0.684185, -1.384026, -2.574885, -0.753478, 1.570796, 2.254981],accel_mss,speed_ms,0,blend_radius_m)
    |   movel([0.685568, -1.382373, -2.576055, -0.753961, 1.570796, 2.256364],accel_mss,speed_ms,0,blend_radius_m)
    |   movel([0.686790, -1.380715, -2.577224, -0.754450, 1.570796, 2.257586],accel_mss,speed_ms,0,blend_radius_m)
    |   movel([0.687866, -1.379044, -2.578399, -0.754946, 1.570796, 2.258662],accel_mss,speed_ms,0,blend_radius_m)
    |   movel([0.688814, -1.377349, -2.579586, -0.755454, 1.570796, 2.259610],accel_mss,speed_ms,0,blend_radius_m)
    |   movel([0.689650, -1.375618, -2.580795, -0.755976, 1.570796, 2.260446],accel_mss,speed_ms,0,blend_radius_m)
    |   movel([0.691053, -1.372013, -2.583298, -0.757078, 1.570796, 2.261849],accel_mss,speed_ms,0,blend_radius_m)
    |   movel([0.685784, -1.377783, -2.579283, -0.755323, 1.570796, 2.256581],accel_mss,speed_ms,0,blend_radius_m)
    |   movel([0.686315, -1.377115, -2.579750, -0.755524, 1.570796, 2.257112],accel_mss,speed_ms,0,blend_radius_m)
    |   movel([0.686734, -1.376414, -2.580240, -0.755735, 1.570796, 2.257530],accel_mss,speed_ms,0,blend_radius_m)
    |   movel([0.687266, -1.374941, -2.581266, -0.756182, 1.570796, 2.258063],accel_mss,speed_ms,0,blend_radius_m)
    |   movel([0.687446, -1.373417, -2.582325, -0.756647, 1.570796, 2.258243],accel_mss,speed_ms,0,blend_radius_m)
    |   movel([0.687344, -1.371902, -2.583375, -0.757112, 1.570796, 2.258140],accel_mss,speed_ms,0,blend_radius_m)
    |   movel([0.687026, -1.370449, -2.584378, -0.757562, 1.570796, 2.257822],accel_mss,speed_ms,0,blend_radius_m)
    |   movel([0.686563, -1.369120, -2.585293, -0.757976, 1.570796, 2.257359],accel_mss,speed_ms,0,blend_radius_m)
    |   movel([0.685474, -1.367060, -2.586706, -0.758623, 1.570796, 2.256271],accel_mss,speed_ms,0,blend_radius_m)
    |   movel([0.684812, -1.370325, -2.584463, -0.757601, 1.570796, 2.255609],accel_mss,speed_ms,0,blend_radius_m)
    |   movel([0.684211, -1.372020, -2.583293, -0.757076, 1.570796, 2.255007],accel_mss,speed_ms,0,blend_radius_m)
    |   movel([0.683325, -1.373573, -2.582217, -0.756599, 1.570796, 2.254122],accel_mss,speed_ms,0,blend_radius_m)
    |   movel([0.682679, -1.373073, -2.582564, -0.756752, 1.570796, 2.253475],accel_mss,speed_ms,0,blend_radius_m)
    |   movel([0.682168, -1.372424, -2.583013, -0.756952, 1.570796, 2.252964],accel_mss,speed_ms,0,blend_radius_m)
    |   movel([0.681364, -1.370863, -2.584092, -0.757434, 1.570796, 2.252160],accel_mss,speed_ms,0,blend_radius_m)
    |   movel([0.680547, -1.369256, -2.585199, -0.757934, 1.570796, 2.251343],accel_mss,speed_ms,0,blend_radius_m)
    |   movel([0.680018, -1.368550, -2.585684, -0.758154, 1.570796, 2.250814],accel_mss,speed_ms,0,blend_radius_m)
    |   movel([0.679351, -1.367971, -2.586082, -0.758336, 1.570796, 2.250148],accel_mss,speed_ms,0,blend_radius_m)
    |   movel([0.677808, -1.369363, -2.585126, -0.757900, 1.570796, 2.248604],accel_mss,speed_ms,0,blend_radius_m)
    |   movel([0.676519, -1.370920, -2.584053, -0.757416, 1.570796, 2.247316],accel_mss,speed_ms,0,blend_radius_m)
    |   movel([0.675488, -1.370319, -2.584467, -0.757603, 1.570796, 2.246284],accel_mss,speed_ms,0,blend_radius_m)
    |   movel([0.674651, -1.369527, -2.585013, -0.757849, 1.570796, 2.245448],accel_mss,speed_ms,0,blend_radius_m)
    |   movel([0.674028, -1.368559, -2.585679, -0.758152, 1.570796, 2.244825],accel_mss,speed_ms,0,blend_radius_m)
    |   movel([0.673638, -1.367440, -2.586446, -0.758503, 1.570796, 2.244435],accel_mss,speed_ms,0,blend_radius_m)
    |   movel([0.673439, -1.367540, -2.586377, -0.758472, 1.570796, 2.244235],accel_mss,speed_ms,0,blend_radius_m)
    |   movel([0.671420, -1.369210, -2.585231, -0.757948, 1.570796, 2.242217],accel_mss,speed_ms,0,blend_radius_m)
    |   movel([0.668987, -1.371379, -2.583736, -0.757274, 1.570796, 2.239783],accel_mss,speed_ms,0,blend_radius_m)
    |   movel([0.667931, -1.372523, -2.582945, -0.756921, 1.570796, 2.238728],accel_mss,speed_ms,0,blend_radius_m)
    |   movel([0.667041, -1.373636, -2.582173, -0.756580, 1.570796, 2.237837],accel_mss,speed_ms,0,blend_radius_m)
    |   movel([0.665423, -1.376052, -2.580492, -0.755845, 1.570796, 2.236220],accel_mss,speed_ms,0,blend_radius_m)
    |   movel([0.664409, -1.371628, -2.583564, -0.757197, 1.570796, 2.235205],accel_mss,speed_ms,0,blend_radius_m)
    |   movel([0.663251, -1.372803, -2.582751, -0.756835, 1.570796, 2.234047],accel_mss,speed_ms,0,blend_radius_m)
    |   movel([0.662173, -1.374044, -2.581890, -0.756455, 1.570796, 2.232970],accel_mss,speed_ms,0,blend_radius_m)
    |   movel([0.660249, -1.376663, -2.580066, -0.755660, 1.570796, 2.231045],accel_mss,speed_ms,0,blend_radius_m)
    |   movel([0.658646, -1.379356, -2.578180, -0.754853, 1.570796, 2.229442],accel_mss,speed_ms,0,blend_radius_m)
    |   movel([0.656967, -1.382805, -2.575749, -0.753835, 1.570796, 2.227763],accel_mss,speed_ms,0,blend_radius_m)
    |   movel([0.656689, -1.383176, -2.575487, -0.753726, 1.570796, 2.227485],accel_mss,speed_ms,0,blend_radius_m)
    |   movel([0.656331, -1.383488, -2.575266, -0.753635, 1.570796, 2.227127],accel_mss,speed_ms,0,blend_radius_m)
    |   movel([0.655764, -1.383746, -2.575083, -0.753560, 1.570796, 2.226561],accel_mss,speed_ms,0,blend_radius_m)
    |   movel([0.652053, -1.384374, -2.574638, -0.753377, 1.570796, 2.222849],accel_mss,speed_ms,0,blend_radius_m)
    |   movel([0.650268, -1.384420, -2.574605, -0.753364, 1.570796, 2.221064],accel_mss,speed_ms,0,blend_radius_m)
    |   movel([0.649684, -1.384265, -2.574715, -0.753409, 1.570796, 2.220481],accel_mss,speed_ms,0,blend_radius_m)
    |   movel([0.649446, -1.383943, -2.574943, -0.753502, 1.570796, 2.220242],accel_mss,speed_ms,0,blend_radius_m)
    |   movel([0.649853, -1.386388, -2.573206, -0.752795, 1.570796, 2.220650],accel_mss,speed_ms,0,blend_radius_m)
    |   movel([0.650227, -1.387521, -2.572398, -0.752470, 1.570796, 2.221024],accel_mss,speed_ms,0,blend_radius_m)
    |   movel([0.650709, -1.388588, -2.571635, -0.752166, 1.570796, 2.221505],accel_mss,speed_ms,0,blend_radius_m)
    |   movel([0.647029, -1.390275, -2.570426, -0.751688, 1.570796, 2.217825],accel_mss,speed_ms,0,blend_radius_m)
    |   movel([0.643033, -1.392287, -2.568978, -0.751124, 1.570796, 2.213829],accel_mss,speed_ms,0,blend_radius_m)
    |   movel([0.641066, -1.393410, -2.568167, -0.750812, 1.570796, 2.211862],accel_mss,speed_ms,0,blend_radius_m)
    |   movel([0.639201, -1.394601, -2.567305, -0.750482, 1.570796, 2.209997],accel_mss,speed_ms,0,blend_radius_m)
    |   movel([0.637498, -1.395863, -2.566390, -0.750136, 1.570796, 2.208294],accel_mss,speed_ms,0,blend_radius_m)
    |   movel([0.636017, -1.397186, -2.565428, -0.749775, 1.570796, 2.206814],accel_mss,speed_ms,0,blend_radius_m)
    |   movel([0.637602, -1.396805, -2.565705, -0.749878, 1.570796, 2.208398],accel_mss,speed_ms,0,blend_radius_m)
    |   movel([0.639142, -1.396591, -2.565861, -0.749937, 1.570796, 2.209939],accel_mss,speed_ms,0,blend_radius_m)
    |   movel([0.640615, -1.396559, -2.565884, -0.749946, 1.570796, 2.211411],accel_mss,speed_ms,0,blend_radius_m)
    |   movel([0.642003, -1.396730, -2.565760, -0.749899, 1.570796, 2.212799],accel_mss,speed_ms,0,blend_radius_m)
    |   movel([0.640831, -1.397176, -2.565436, -0.749778, 1.570796, 2.211628],accel_mss,speed_ms,0,blend_radius_m)
    |   movel([0.638537, -1.398337, -2.564589, -0.749463, 1.570796, 2.209333],accel_mss,speed_ms,0,blend_radius_m)
    |   movel([0.637430, -1.399041, -2.564075, -0.749273, 1.570796, 2.208227],accel_mss,speed_ms,0,blend_radius_m)
    |   movel([0.635360, -1.400650, -2.562897, -0.748842, 1.570796, 2.206157],accel_mss,speed_ms,0,blend_radius_m)
    |   movel([0.634413, -1.401543, -2.562241, -0.748605, 1.570796, 2.205210],accel_mss,speed_ms,0,blend_radius_m)
    |   movel([0.633542, -1.402484, -2.561549, -0.748356, 1.570796, 2.204338],accel_mss,speed_ms,0,blend_radius_m)
    |   speed_ms = 0.005
    |   movel([0.633542, -1.393830, -2.557656, -0.760903, 1.570796, 2.204338],accel_mss,speed_ms,0,blend_radius_m)
    |   speed_ms = 0.040
    |   movel([0.636386, -1.399066, -2.553833, -0.759490, 1.570796, 2.207182],accel_mss,speed_ms,0,blend_radius_m)
    |   speed_ms = 0.005
    |   movel([0.636386, -1.407681, -2.557704, -0.747004, 1.570796, 2.207182],accel_mss,speed_ms,0,blend_radius_m)
    |   speed_ms = 0.025
    |   movel([0.637314, -1.406280, -2.558745, -0.747364, 1.570796, 2.208111],accel_mss,speed_ms,0,blend_radius_m)
    |   movel([0.638362, -1.404895, -2.559771, -0.747724, 1.570796, 2.209158],accel_mss,speed_ms,0,blend_radius_m)
    |   movel([0.639519, -1.403542, -2.560770, -0.748077, 1.570796, 2.210315],accel_mss,speed_ms,0,blend_radius_m)
    |   movel([0.640773, -1.402239, -2.561729, -0.748420, 1.570796, 2.211570],accel_mss,speed_ms,0,blend_radius_m)
    |   movel([0.642119, -1.401000, -2.562640, -0.748749, 1.570796, 2.212915],accel_mss,speed_ms,0,blend_radius_m)
    |   movel([0.643542, -1.399840, -2.563490, -0.749059, 1.570796, 2.214339],accel_mss,speed_ms,0,blend_radius_m)
    |   movel([0.645035, -1.398773, -2.564271, -0.749345, 1.570796, 2.215832],accel_mss,speed_ms,0,blend_radius_m)
    |   movel([0.646587, -1.397817, -2.564968, -0.749604, 1.570796, 2.217384],accel_mss,speed_ms,0,blend_radius_m)
    |   movel([0.651504, -1.395060, -2.566973, -0.750356, 1.570796, 2.222301],accel_mss,speed_ms,0,blend_radius_m)
    |   movel([0.652584, -1.394320, -2.567509, -0.750560, 1.570796, 2.223380],accel_mss,speed_ms,0,blend_radius_m)
    |   movel([0.653628, -1.393474, -2.568121, -0.750794, 1.570796, 2.224424],accel_mss,speed_ms,0,blend_radius_m)
    |   movel([0.654647, -1.392483, -2.568837, -0.751069, 1.570796, 2.225443],accel_mss,speed_ms,0,blend_radius_m)
    |   movel([0.655657, -1.391300, -2.569689, -0.751400, 1.570796, 2.226453],accel_mss,speed_ms,0,blend_radius_m)
    |   movel([0.658245, -1.387723, -2.572253, -0.752412, 1.570796, 2.229042],accel_mss,speed_ms,0,blend_radius_m)
    |   movel([0.659612, -1.385970, -2.573503, -0.752915, 1.570796, 2.230408],accel_mss,speed_ms,0,blend_radius_m)
    |   movel([0.661189, -1.384329, -2.574670, -0.753390, 1.570796, 2.231986],accel_mss,speed_ms,0,blend_radius_m)
    |   movel([0.662268, -1.383437, -2.575302, -0.753650, 1.570796, 2.233065],accel_mss,speed_ms,0,blend_radius_m)
    |   movel([0.663410, -1.382641, -2.575865, -0.753883, 1.570796, 2.234206],accel_mss,speed_ms,0,blend_radius_m)
    |   movel([0.665831, -1.381298, -2.576813, -0.754277, 1.570796, 2.236627],accel_mss,speed_ms,0,blend_radius_m)
    |   movel([0.668358, -1.380204, -2.577584, -0.754601, 1.570796, 2.239154],accel_mss,speed_ms,0,blend_radius_m)
    |   movel([0.670899, -1.379264, -2.578245, -0.754881, 1.570796, 2.241695],accel_mss,speed_ms,0,blend_radius_m)
    |   movel([0.673349, -1.378439, -2.578823, -0.755127, 1.570796, 2.244146],accel_mss,speed_ms,0,blend_radius_m)
    |   movel([0.675779, -1.377820, -2.579257, -0.755312, 1.570796, 2.246575],accel_mss,speed_ms,0,blend_radius_m)
    |   movel([0.676936, -1.377654, -2.579373, -0.755362, 1.570796, 2.247732],accel_mss,speed_ms,0,blend_radius_m)
    |   movel([0.678032, -1.377616, -2.579400, -0.755373, 1.570796, 2.248829],accel_mss,speed_ms,0,blend_radius_m)
    |   movel([0.679041, -1.377734, -2.579317, -0.755338, 1.570796, 2.249838],accel_mss,speed_ms,0,blend_radius_m)
    |   movel([0.679953, -1.378031, -2.579109, -0.755249, 1.570796, 2.250749],accel_mss,speed_ms,0,blend_radius_m)
    |   speed_ms = 0.005
    |   movel([0.679953, -1.369198, -2.575109, -0.768082, 1.570796, 2.250749],accel_mss,speed_ms,0,blend_radius_m)
    |   speed_ms = 0.040
    |   movel([0.680324, -1.370938, -2.573904, -0.767547, 1.570796, 2.251120],accel_mss,speed_ms,0,blend_radius_m)
    |   speed_ms = 0.005
    |   movel([0.680324, -1.379759, -2.577897, -0.754733, 1.570796, 2.251120],accel_mss,speed_ms,0,blend_radius_m)
    |   speed_ms = 0.025
    |   movel([0.680472, -1.380248, -2.577553, -0.754588, 1.570796, 2.251269],accel_mss,speed_ms,0,blend_radius_m)
    |   movel([0.680607, -1.381026, -2.577005, -0.754358, 1.570796, 2.251403],accel_mss,speed_ms,0,blend_radius_m)
    |   movel([0.680415, -1.382962, -2.575638, -0.753789, 1.570796, 2.251212],accel_mss,speed_ms,0,blend_radius_m)
    |   movel([0.680140, -1.383978, -2.574919, -0.753492, 1.570796, 2.250936],accel_mss,speed_ms,0,blend_radius_m)
    |   movel([0.679886, -1.384452, -2.574583, -0.753355, 1.570796, 2.250682],accel_mss,speed_ms,0,blend_radius_m)
    |   movel([0.679748, -1.384511, -2.574541, -0.753337, 1.570796, 2.250544],accel_mss,speed_ms,0,blend_radius_m)
    |   movel([0.679605, -1.384387, -2.574628, -0.753373, 1.570796, 2.250401],accel_mss,speed_ms,0,blend_radius_m)
    |   movel([0.678556, -1.382444, -2.576005, -0.753941, 1.570796, 2.249352],accel_mss,speed_ms,0,blend_radius_m)
    |   movel([0.677827, -1.381621, -2.576586, -0.754182, 1.570796, 2.248623],accel_mss,speed_ms,0,blend_radius_m)
    |   movel([0.677344, -1.381336, -2.576787, -0.754266, 1.570796, 2.248140],accel_mss,speed_ms,0,blend_radius_m)
    |   movel([0.676759, -1.381163, -2.576909, -0.754317, 1.570796, 2.247556],accel_mss,speed_ms,0,blend_radius_m)
    |   movel([0.676002, -1.381140, -2.576925, -0.754324, 1.570796, 2.246799],accel_mss,speed_ms,0,blend_radius_m)
    |   movel([0.675193, -1.381241, -2.576854, -0.754294, 1.570796, 2.245989],accel_mss,speed_ms,0,blend_radius_m)
    |   movel([0.673139, -1.381692, -2.576535, -0.754161, 1.570796, 2.243936],accel_mss,speed_ms,0,blend_radius_m)
    |   movel([0.671022, -1.382358, -2.576065, -0.753966, 1.570796, 2.241819],accel_mss,speed_ms,0,blend_radius_m)
    |   movel([0.668907, -1.383214, -2.575460, -0.753715, 1.570796, 2.239703],accel_mss,speed_ms,0,blend_radius_m)
    |   movel([0.666865, -1.384233, -2.574738, -0.753418, 1.570796, 2.237662],accel_mss,speed_ms,0,blend_radius_m)
    |   movel([0.666548, -1.386886, -2.572851, -0.752652, 1.570796, 2.237345],accel_mss,speed_ms,0,blend_radius_m)
    |   movel([0.665908, -1.389602, -2.570908, -0.751878, 1.570796, 2.236704],accel_mss,speed_ms,0,blend_radius_m)
    |   movel([0.665535, -1.388831, -2.571461, -0.752097, 1.570796, 2.236331],accel_mss,speed_ms,0,blend_radius_m)
    |   movel([0.664970, -1.388198, -2.571914, -0.752277, 1.570796, 2.235766],accel_mss,speed_ms,0,blend_radius_m)
    |   movel([0.664228, -1.387728, -2.572250, -0.752411, 1.570796, 2.235024],accel_mss,speed_ms,0,blend_radius_m)
    |   movel([0.663335, -1.387437, -2.572458, -0.752494, 1.570796, 2.234131],accel_mss,speed_ms,0,blend_radius_m)
    |   movel([0.662824, -1.387478, -2.572429, -0.752482, 1.570796, 2.233620],accel_mss,speed_ms,0,blend_radius_m)
    |   movel([0.662439, -1.387841, -2.572169, -0.752379, 1.570796, 2.233236],accel_mss,speed_ms,0,blend_radius_m)
    |   movel([0.659039, -1.392277, -2.568985, -0.751127, 1.570796, 2.229836],accel_mss,speed_ms,0,blend_radius_m)
    |   movel([0.657166, -1.394455, -2.567412, -0.750523, 1.570796, 2.227962],accel_mss,speed_ms,0,blend_radius_m)
    |   movel([0.655132, -1.396589, -2.565863, -0.749938, 1.570796, 2.225928],accel_mss,speed_ms,0,blend_radius_m)
    |   movel([0.652972, -1.398610, -2.564390, -0.749389, 1.570796, 2.223768],accel_mss,speed_ms,0,blend_radius_m)
    |   movel([0.650715, -1.400452, -2.563042, -0.748895, 1.570796, 2.221511],accel_mss,speed_ms,0,blend_radius_m)
    |   movel([0.646073, -1.404040, -2.560402, -0.747947, 1.570796, 2.216869],accel_mss,speed_ms,0,blend_radius_m)
    |   movel([0.643941, -1.405968, -2.558976, -0.747445, 1.570796, 2.214738],accel_mss,speed_ms,0,blend_radius_m)
    |   movel([0.642036, -1.408099, -2.557393, -0.746897, 1.570796, 2.212832],accel_mss,speed_ms,0,blend_radius_m)
    |   speed_ms = 0.005
    |   movel([0.642036, -1.399487, -2.553524, -0.759378, 1.570796, 2.212832],accel_mss,speed_ms,0,blend_radius_m)
    |   speed_ms = 0.040
    |   movel([0.652406, -1.400382, -2.552866, -0.759141, 1.570796, 2.223202],accel_mss,speed_ms,0,blend_radius_m)
    |   speed_ms = 0.005
    |   movel([0.652406, -1.408988, -2.556731, -0.746670, 1.570796, 2.223202],accel_mss,speed_ms,0,blend_radius_m)
    |   speed_ms = 0.025
    |   movel([0.650892, -1.410707, -2.555447, -0.746235, 1.570796, 2.221688],accel_mss,speed_ms,0,blend_radius_m)
    |   movel([0.649148, -1.412267, -2.554278, -0.745844, 1.570796, 2.219944],accel_mss,speed_ms,0,blend_radius_m)
